LIN {X 0,Y 532.291,Z 792.488,A -85,B 0,C 180,E1 -4217.451,E2 -4217.451} C_VEL
LIN {X 0,Y 532.141,Z 804.373,A -85,B 0,C 180,E1 -4218.078,E2 -4218.078} C_VEL
LIN {X 0,Y 531.859,Z 815.786,A -85,B 0,C 180,E1 -4218.853,E2 -4218.853} C_VEL
LIN {X 0,Y 531.632,Z 825.925,A -85,B 0,C 180,E1 -4219.715,E2 -4219.715} C_VEL
LIN {X 0,Y 531.41,Z 835.007,A -85,B 0,C 180,E1 -4220.672,E2 -4220.672} C_VEL
LIN {X 0,Y 531.158,Z 843.796,A -85,B 0,C 180,E1 -4221.818,E2 -4221.818} C_VEL
LIN {X 0,Y 530.974,Z 851.482,A -85,B 0,C 180,E1 -4223.077,E2 -4223.077} C_VEL
LIN {X 0,Y 530.875,Z 857.285,A -85,B 0,C 180,E1 -4224.297,E2 -4224.297} C_VEL
LIN {X 0,Y 530.745,Z 861.535,A -85,B 0,C 180,E1 -4225.438,E2 -4225.438} C_VEL
LIN {X 0,Y 530.706,Z 863.774,A -85,B 0,C 180,E1 -4226.199,E2 -4226.199} C_VEL
LIN {X 0,Y 530.655,Z 865.602,A -85,B 0,C 180,E1 -4226.958,E2 -4226.958} C_VEL
LIN {X 0,Y 530.61,Z 866.987,A -85,B 0,C 180,E1 -4227.718,E2 -4227.718} C_VEL
LIN {X 0,Y 530.592,Z 868.572,A -85,B 0,C 180,E1 -4229.236,E2 -4229.236} C_VEL
LIN {X 0,Y 530.583,Z 868.809,A -85,B 0,C 180,E1 -4229.995,E2 -4229.995} C_VEL
LIN {X 0,Y 530.623,Z 868.067,A -85,B 0,C 180,E1 -4231.513,E2 -4231.513} C_VEL
LIN {X 0,Y 530.65,Z 865.813,A -85,B 0,C 180,E1 -4233.032,E2 -4233.032} C_VEL
LIN {X 0,Y 530.738,Z 863.013,A -85,B 0,C 180,E1 -4234.171,E2 -4234.171} C_VEL
LIN {X 0,Y 530.785,Z 859.223,A -85,B 0,C 180,E1 -4235.313,E2 -4235.313} C_VEL
LIN {X 0,Y 530.93,Z 853.861,A -85,B 0,C 180,E1 -4236.551,E2 -4236.551} C_VEL
LIN {X 0,Y 531.084,Z 846.949,A -85,B 0,C 180,E1 -4237.79,E2 -4237.79} C_VEL
LIN {X 0,Y 531.313,Z 838.946,A -85,B 0,C 180,E1 -4238.936,E2 -4238.936} C_VEL
LIN {X 0,Y 531.519,Z 830.744,A -85,B 0,C 180,E1 -4239.892,E2 -4239.892} C_VEL
LIN {X 0,Y 531.753,Z 820.601,A -85,B 0,C 180,E1 -4240.85,E2 -4240.85} C_VEL
LIN {X 0,Y 532.059,Z 810.192,A -85,B 0,C 180,E1 -4241.638,E2 -4241.638} C_VEL
LIN {X 0,Y 532.239,Z 798.418,A -85,B 0,C 180,E1 -4242.348,E2 -4242.348} C_VEL
LIN {X 0,Y 532.349,Z 785.959,A -85,B 0,C 180,E1 -4242.91,E2 -4242.91} C_VEL
LIN {X 0,Y 532.464,Z 772.907,A -85,B 0,C 180,E1 -4243.325,E2 -4243.325} C_VEL
LIN {X 0,Y 532.541,Z 760.671,A -85,B 0,C 180,E1 -4243.566,E2 -4243.566} C_VEL
LIN {X 0,Y 532.699,Z 691.55,A -85,B 0,C 180,E1 -4244.506,E2 -4244.506} C_VEL
LIN {X 0,Y 531.049,Z 686.337,A -85,B 0,C 180,E1 -4244.639,E2 -4244.639} C_VEL
LIN {X 0,Y 530.967,Z 686.343,A -85,B 0,C 180,E1 -4247.718,E2 -4247.718} C_VEL
LIN {X 0,Y 531.008,Z 686.337,A -85,B 0,C 180,E1 -4250.121,E2 -4250.121} C_VEL
LIN {X 0,Y 530.923,Z 686.348,A -85,B 0,C 180,E1 -4252.567,E2 -4252.567} C_VEL
LIN {X 0,Y 530.945,Z 686.35,A -85,B 0,C 180,E1 -4255.053,E2 -4255.053} C_VEL
LIN {X 0,Y 530.984,Z 686.34,A -85,B 0,C 180,E1 -4257.589,E2 -4257.589} C_VEL
LIN {X 0,Y 530.943,Z 686.344,A -85,B 0,C 180,E1 -4260.639,E2 -4260.639} C_VEL
LIN {X 0,Y 530.955,Z 686.344,A -85,B 0,C 180,E1 -4263.766,E2 -4263.766} C_VEL
LIN {X 0,Y 530.927,Z 686.345,A -85,B 0,C 180,E1 -4266.552,E2 -4266.552} C_VEL
LIN {X 0,Y 530.964,Z 686.345,A -85,B 0,C 180,E1 -4269.851,E2 -4269.851} C_VEL
LIN {X 0,Y 530.941,Z 686.344,A -85,B 0,C 180,E1 -4272.45,E2 -4272.45} C_VEL
LIN {X 0,Y 530.937,Z 686.346,A -85,B 0,C 180,E1 -4275.615,E2 -4275.615} C_VEL
LIN {X 0,Y 530.968,Z 686.341,A -85,B 0,C 180,E1 -4278.562,E2 -4278.562} C_VEL
LIN {X 0,Y 530.97,Z 686.339,A -85,B 0,C 180,E1 -4280.555,E2 -4280.555} C_VEL
LIN {X 0,Y 530.915,Z 686.355,A -85,B 0,C 180,E1 -4283.837,E2 -4283.837} C_VEL
LIN {X 0,Y 530.938,Z 686.345,A -85,B 0,C 180,E1 -4286.489,E2 -4286.489} C_VEL
LIN {X 0,Y 530.946,Z 686.342,A -85,B 0,C 180,E1 -4289.344,E2 -4289.344} C_VEL
LIN {X 0,Y 530.953,Z 686.347,A -85,B 0,C 180,E1 -4292.462,E2 -4292.462} C_VEL
LIN {X 0,Y 530.958,Z 686.341,A -85,B 0,C 180,E1 -4294.94,E2 -4294.94} C_VEL
LIN {X 0,Y 530.91,Z 686.353,A -85,B 0,C 180,E1 -4298.244,E2 -4298.244} C_VEL
LIN {X 0,Y 530.925,Z 686.349,A -85,B 0,C 180,E1 -4300.675,E2 -4300.675} C_VEL
LIN {X 0,Y 530.926,Z 686.344,A -85,B 0,C 180,E1 -4303.069,E2 -4303.069} C_VEL
LIN {X 0,Y 530.975,Z 686.339,A -85,B 0,C 180,E1 -4305.435,E2 -4305.435} C_VEL
LIN {X 0,Y 530.983,Z 686.345,A -85,B 0,C 180,E1 -4308.548,E2 -4308.548} C_VEL
LIN {X 0,Y 530.989,Z 686.337,A -85,B 0,C 180,E1 -4311.628,E2 -4311.628} C_VEL
LIN {X 0,Y 531.075,Z 686.334,A -85,B 0,C 180,E1 -4314.685,E2 -4314.685} C_VEL
LIN {X 0,Y 531.061,Z 686.328,A -85,B 0,C 180,E1 -4317.725,E2 -4317.725} C_VEL
LIN {X 0,Y 531.084,Z 686.332,A -85,B 0,C 180,E1 -4320.758,E2 -4320.758} C_VEL
LIN {X 0,Y 531.043,Z 686.337,A -85,B 0,C 180,E1 -4323.034,E2 -4323.034} C_VEL
LIN {X 0,Y 531.015,Z 686.335,A -85,B 0,C 180,E1 -4326.078,E2 -4326.078} C_VEL
LIN {X 0,Y 530.969,Z 686.346,A -85,B 0,C 180,E1 -4329.139,E2 -4329.139} C_VEL
LIN {X 0,Y 530.989,Z 686.342,A -85,B 0,C 180,E1 -4331.683,E2 -4331.683} C_VEL
LIN {X 0,Y 530.972,Z 686.342,A -85,B 0,C 180,E1 -4334.966,E2 -4334.966} C_VEL
LIN {X 0,Y 530.944,Z 686.349,A -85,B 0,C 180,E1 -4337.725,E2 -4337.725} C_VEL
LIN {X 0,Y 530.933,Z 686.342,A -85,B 0,C 180,E1 -4340.941,E2 -4340.941} C_VEL
LIN {X 0,Y 530.958,Z 686.342,A -85,B 0,C 180,E1 -4344.226,E2 -4344.226} C_VEL
LIN {X 0,Y 530.956,Z 686.34,A -85,B 0,C 180,E1 -4346.746,E2 -4346.746} C_VEL
LIN {X 0,Y 530.935,Z 686.345,A -85,B 0,C 180,E1 -4349.326,E2 -4349.326} C_VEL
LIN {X 0,Y 530.92,Z 686.353,A -85,B 0,C 180,E1 -4352.108,E2 -4352.108} C_VEL
LIN {X 0,Y 530.93,Z 686.344,A -85,B 0,C 180,E1 -4354.859,E2 -4354.859} C_VEL
LIN {X 0,Y 530.911,Z 686.348,A -85,B 0,C 180,E1 -4357.512,E2 -4357.512} C_VEL
LIN {X 0,Y 530.981,Z 686.344,A -85,B 0,C 180,E1 -4360.433,E2 -4360.433} C_VEL
LIN {X 0,Y 530.917,Z 686.347,A -85,B 0,C 180,E1 -4363.5,E2 -4363.5} C_VEL
LIN {X 0,Y 530.918,Z 686.352,A -85,B 0,C 180,E1 -4366.511,E2 -4366.511} C_VEL
LIN {X 0,Y 530.966,Z 686.341,A -85,B 0,C 180,E1 -4369.576,E2 -4369.576} C_VEL
LIN {X 0,Y 530.928,Z 686.353,A -85,B 0,C 180,E1 -4372.583,E2 -4372.583} C_VEL
LIN {X 0,Y 530.962,Z 686.34,A -85,B 0,C 180,E1 -4375.317,E2 -4375.317} C_VEL
LIN {X 0,Y 530.934,Z 686.348,A -85,B 0,C 180,E1 -4378.038,E2 -4378.038} C_VEL
LIN {X 0,Y 530.962,Z 686.35,A -85,B 0,C 180,E1 -4381.139,E2 -4381.139} C_VEL
LIN {X 0,Y 531.008,Z 686.532,A -85,B 0,C 180,E1 -4381.45,E2 -4381.45} C_VEL
LIN {X 0,Y 533.727,Z 698.362,A -85,B 0,C 180,E1 -4382.988,E2 -4382.988} C_VEL
LIN {X 0,Y 533.507,Z 718.499,A -85,B 0,C 180,E1 -4385.361,E2 -4385.361} C_VEL
LIN {X 0,Y 532.997,Z 742.504,A -85,B 0,C 180,E1 -4388.137,E2 -4388.137} C_VEL
LIN {X 0,Y 532.397,Z 768.598,A -85,B 0,C 180,E1 -4391.137,E2 -4391.137} C_VEL
LIN {X 0,Y 531.853,Z 792.13,A -85,B 0,C 180,E1 -4393.895,E2 -4393.895} C_VEL
LIN {X 0,Y 531.68,Z 801.876,A -85,B 0,C 180,E1 -4395.029,E2 -4395.029} C_VEL
LIN {X 0,Y 532.81,Z 811.855,A -85,B 0,C 180,E1 -4395.201,E2 -4395.201} C_VEL
LIN {X 0,Y 532.375,Z 912.231,A -85,B 0,C 180,E1 -4396.576,E2 -4396.576} C_VEL
LIN {X 0,Y 532.216,Z 925.399,A -85,B 0,C 180,E1 -4396.912,E2 -4396.912} C_VEL
LIN {X 0,Y 531.975,Z 937.504,A -85,B 0,C 180,E1 -4397.367,E2 -4397.367} C_VEL
LIN {X 0,Y 531.811,Z 948.839,A -85,B 0,C 180,E1 -4397.94,E2 -4397.94} C_VEL
LIN {X 0,Y 531.567,Z 959.985,A -85,B 0,C 180,E1 -4398.664,E2 -4398.664} C_VEL
LIN {X 0,Y 531.26,Z 970.602,A -85,B 0,C 180,E1 -4399.526,E2 -4399.526} C_VEL
LIN {X 0,Y 531.062,Z 980.153,A -85,B 0,C 180,E1 -4400.484,E2 -4400.484} C_VEL
LIN {X 0,Y 530.885,Z 988.003,A -85,B 0,C 180,E1 -4401.441,E2 -4401.441} C_VEL
LIN {X 0,Y 530.684,Z 995.655,A -85,B 0,C 180,E1 -4402.587,E2 -4402.587} C_VEL
LIN {X 0,Y 530.599,Z 1002.705,A -85,B 0,C 180,E1 -4403.923,E2 -4403.923} C_VEL
LIN {X 0,Y 530.457,Z 1007.392,A -85,B 0,C 180,E1 -4405.065,E2 -4405.065} C_VEL
LIN {X 0,Y 530.514,Z 1010.975,A -85,B 0,C 180,E1 -4406.207,E2 -4406.207} C_VEL
LIN {X 0,Y 530.456,Z 1012.821,A -85,B 0,C 180,E1 -4406.967,E2 -4406.967} C_VEL
LIN {X 0,Y 530.409,Z 1014.205,A -85,B 0,C 180,E1 -4407.727,E2 -4407.727} C_VEL
LIN {X 0,Y 530.344,Z 1015.789,A -85,B 0,C 180,E1 -4409.246,E2 -4409.246} C_VEL
LIN {X 0,Y 530.342,Z 1016,A -85,B 0,C 180,E1 -4410.005,E2 -4410.005} C_VEL
LIN {X 0,Y 530.361,Z 1015.178,A -85,B 0,C 180,E1 -4411.524,E2 -4411.524} C_VEL
LIN {X 0,Y 530.411,Z 1014.188,A -85,B 0,C 180,E1 -4412.283,E2 -4412.283} C_VEL
LIN {X 0,Y 530.458,Z 1012.797,A -85,B 0,C 180,E1 -4413.043,E2 -4413.043} C_VEL
LIN {X 0,Y 530.524,Z 1009.881,A -85,B 0,C 180,E1 -4414.183,E2 -4414.183} C_VEL
LIN {X 0,Y 530.526,Z 1005.932,A -85,B 0,C 180,E1 -4415.325,E2 -4415.325} C_VEL
LIN {X 0,Y 530.604,Z 1000.238,A -85,B 0,C 180,E1 -4416.587,E2 -4416.587} C_VEL
LIN {X 0,Y 530.763,Z 993.207,A -85,B 0,C 180,E1 -4417.805,E2 -4417.805} C_VEL
LIN {X 0,Y 530.932,Z 984.957,A -85,B 0,C 180,E1 -4418.952,E2 -4418.952} C_VEL
LIN {X 0,Y 531.112,Z 976.496,A -85,B 0,C 180,E1 -4419.91,E2 -4419.91} C_VEL
LIN {X 0,Y 531.415,Z 966.041,A -85,B 0,C 180,E1 -4420.867,E2 -4420.867} C_VEL
LIN {X 0,Y 531.648,Z 955.001,A -85,B 0,C 180,E1 -4421.681,E2 -4421.681} C_VEL
LIN {X 0,Y 531.912,Z 944.33,A -85,B 0,C 180,E1 -4422.306,E2 -4422.306} C_VEL
LIN {X 0,Y 532.097,Z 932.66,A -85,B 0,C 180,E1 -4422.834,E2 -4422.834} C_VEL
LIN {X 0,Y 532.285,Z 919.192,A -85,B 0,C 180,E1 -4423.267,E2 -4423.267} C_VEL
LIN {X 0,Y 532.452,Z 905.789,A -85,B 0,C 180,E1 -4423.53,E2 -4423.53} C_VEL
LIN {X 0,Y 532.775,Z 810.11,A -85,B 0,C 180,E1 -4424.824,E2 -4424.824} C_VEL
LIN {X 0,Y 531.69,Z 801.879,A -85,B 0,C 180,E1 -4424.97,E2 -4424.97} C_VEL
LIN {X 0,Y 532.296,Z 774.205,A -85,B 0,C 180,E1 -4428.201,E2 -4428.201} C_VEL
LIN {X 0,Y 532.732,Z 753.381,A -85,B 0,C 180,E1 -4430.62,E2 -4430.62} C_VEL
LIN {X 0,Y 533.236,Z 730.084,A -85,B 0,C 180,E1 -4433.294,E2 -4433.294} C_VEL
LIN {X 0,Y 533.69,Z 705.785,A -85,B 0,C 180,E1 -4436.131,E2 -4436.131} C_VEL
LIN {X 0,Y 533.739,Z 698.273,A -85,B 0,C 180,E1 -4437.022,E2 -4437.022} C_VEL
LIN {X 0,Y 530.97,Z 686.348,A -85,B 0,C 180,E1 -4438.587,E2 -4438.587} C_VEL
LIN {X 0,Y 530.938,Z 686.353,A -85,B 0,C 180,E1 -4441.084,E2 -4441.084} C_VEL
LIN {X 0,Y 530.897,Z 686.353,A -85,B 0,C 180,E1 -4443.783,E2 -4443.783} C_VEL
LIN {X 0,Y 530.902,Z 686.347,A -85,B 0,C 180,E1 -4446.566,E2 -4446.566} C_VEL
LIN {X 0,Y 530.941,Z 686.349,A -85,B 0,C 180,E1 -4449.451,E2 -4449.451} C_VEL
LIN {X 0,Y 530.917,Z 686.347,A -85,B 0,C 180,E1 -4452.466,E2 -4452.466} C_VEL
LIN {X 0,Y 530.974,Z 686.345,A -85,B 0,C 180,E1 -4455.451,E2 -4455.451} C_VEL
LIN {X 0,Y 530.965,Z 686.342,A -85,B 0,C 180,E1 -4458.561,E2 -4458.561} C_VEL
LIN {X 0,Y 530.96,Z 686.347,A -85,B 0,C 180,E1 -4461.529,E2 -4461.529} C_VEL
LIN {X 0,Y 530.948,Z 686.343,A -85,B 0,C 180,E1 -4464.379,E2 -4464.379} C_VEL
LIN {X 0,Y 530.979,Z 686.346,A -85,B 0,C 180,E1 -4467.134,E2 -4467.134} C_VEL
LIN {X 0,Y 530.965,Z 686.344,A -85,B 0,C 180,E1 -4469.803,E2 -4469.803} C_VEL
LIN {X 0,Y 530.977,Z 686.341,A -85,B 0,C 180,E1 -4472.478,E2 -4472.478} C_VEL
LIN {X 0,Y 530.989,Z 686.342,A -85,B 0,C 180,E1 -4474.942,E2 -4474.942} C_VEL
LIN {X 0,Y 530.982,Z 686.34,A -85,B 0,C 180,E1 -4478.247,E2 -4478.247} C_VEL
LIN {X 0,Y 531.001,Z 686.339,A -85,B 0,C 180,E1 -4480.677,E2 -4480.677} C_VEL
LIN {X 0,Y 530.974,Z 686.346,A -85,B 0,C 180,E1 -4483.071,E2 -4483.071} C_VEL
LIN {X 0,Y 531.031,Z 686.341,A -85,B 0,C 180,E1 -4485.534,E2 -4485.534} C_VEL
LIN {X 0,Y 532.595,Z 691.472,A -85,B 0,C 180,E1 -4485.655,E2 -4485.655} C_VEL
LIN {X 0,Y 532.362,Z 763.672,A -85,B 0,C 180,E1 -4486.667,E2 -4486.667} C_VEL
LIN {X 0,Y 532.273,Z 775.605,A -85,B 0,C 180,E1 -4486.956,E2 -4486.956} C_VEL
LIN {X 0,Y 532.095,Z 785.975,A -85,B 0,C 180,E1 -4487.315,E2 -4487.315} C_VEL
LIN {X 0,Y 531.937,Z 796.416,A -85,B 0,C 180,E1 -4487.796,E2 -4487.796} C_VEL
LIN {X 0,Y 531.787,Z 805.876,A -85,B 0,C 180,E1 -4488.344,E2 -4488.344} C_VEL
LIN {X 0,Y 531.527,Z 815.647,A -85,B 0,C 180,E1 -4489.043,E2 -4489.043} C_VEL
LIN {X 0,Y 531.372,Z 823.465,A -85,B 0,C 180,E1 -4489.715,E2 -4489.715} C_VEL
LIN {X 0,Y 531.113,Z 832.637,A -85,B 0,C 180,E1 -4490.671,E2 -4490.671} C_VEL
LIN {X 0,Y 530.923,Z 840.17,A -85,B 0,C 180,E1 -4491.627,E2 -4491.627} C_VEL
LIN {X 0,Y 530.792,Z 846.415,A -85,B 0,C 180,E1 -4492.583,E2 -4492.583} C_VEL
LIN {X 0,Y 530.69,Z 852.318,A -85,B 0,C 180,E1 -4493.686,E2 -4493.686} C_VEL
LIN {X 0,Y 530.581,Z 856.628,A -85,B 0,C 180,E1 -4494.68,E2 -4494.68} C_VEL
LIN {X 0,Y 530.562,Z 860.504,A -85,B 0,C 180,E1 -4495.822,E2 -4495.822} C_VEL
LIN {X 0,Y 530.499,Z 863.37,A -85,B 0,C 180,E1 -4496.962,E2 -4496.962} C_VEL
LIN {X 0,Y 530.43,Z 864.833,A -85,B 0,C 180,E1 -4497.722,E2 -4497.722} C_VEL
LIN {X 0,Y 530.375,Z 866.384,A -85,B 0,C 180,E1 -4499.241,E2 -4499.241} C_VEL
LIN {X 0,Y 530.371,Z 866.629,A -85,B 0,C 180,E1 -4500,E2 -4500} C_VEL
LIN {X 0,Y 530.384,Z 865.83,A -85,B 0,C 180,E1 -4501.519,E2 -4501.519} C_VEL
LIN {X 0,Y 530.425,Z 864.921,A -85,B 0,C 180,E1 -4502.278,E2 -4502.278} C_VEL
LIN {X 0,Y 530.55,Z 861.742,A -85,B 0,C 180,E1 -4503.798,E2 -4503.798} C_VEL
LIN {X 0,Y 530.524,Z 858.271,A -85,B 0,C 180,E1 -4504.94,E2 -4504.94} C_VEL
LIN {X 0,Y 530.669,Z 853.695,A -85,B 0,C 180,E1 -4506.082,E2 -4506.082} C_VEL
LIN {X 0,Y 530.754,Z 847.914,A -85,B 0,C 180,E1 -4507.227,E2 -4507.227} C_VEL
LIN {X 0,Y 530.91,Z 841.981,A -85,B 0,C 180,E1 -4508.181,E2 -4508.181} C_VEL
LIN {X 0,Y 531.06,Z 834.829,A -85,B 0,C 180,E1 -4509.138,E2 -4509.138} C_VEL
LIN {X 0,Y 531.292,Z 826.099,A -85,B 0,C 180,E1 -4510.095,E2 -4510.095} C_VEL
LIN {X 0,Y 531.474,Z 816.505,A -85,B 0,C 180,E1 -4510.958,E2 -4510.958} C_VEL
LIN {X 0,Y 531.733,Z 807.033,A -85,B 0,C 180,E1 -4511.653,E2 -4511.653} C_VEL
LIN {X 0,Y 531.927,Z 797.845,A -85,B 0,C 180,E1 -4512.204,E2 -4512.204} C_VEL
LIN {X 0,Y 532.049,Z 787.908,A -85,B 0,C 180,E1 -4512.686,E2 -4512.686} C_VEL
LIN {X 0,Y 532.22,Z 777.605,A -85,B 0,C 180,E1 -4513.07,E2 -4513.07} C_VEL
LIN {X 0,Y 532.354,Z 767.993,A -85,B 0,C 180,E1 -4513.334,E2 -4513.334} C_VEL
LIN {X 0,Y 532.42,Z 756.137,A -85,B 0,C 180,E1 -4513.551,E2 -4513.551} C_VEL
LIN {X 0,Y 532.573,Z 691.328,A -85,B 0,C 180,E1 -4514.441,E2 -4514.441} C_VEL
LIN {X 0,Y 531.088,Z 686.334,A -85,B 0,C 180,E1 -4514.562,E2 -4514.562} C_VEL
LIN {X 0,Y 530.993,Z 686.338,A -85,B 0,C 180,E1 -4517.723,E2 -4517.723} C_VEL
LIN {X 0,Y 531.026,Z 686.334,A -85,B 0,C 180,E1 -4520.127,E2 -4520.127} C_VEL
LIN {X 0,Y 530.954,Z 686.348,A -85,B 0,C 180,E1 -4522.573,E2 -4522.573} C_VEL
LIN {X 0,Y 530.99,Z 686.343,A -85,B 0,C 180,E1 -4525.059,E2 -4525.059} C_VEL
LIN {X 0,Y 530.977,Z 686.338,A -85,B 0,C 180,E1 -4527.598,E2 -4527.598} C_VEL
LIN {X 0,Y 530.973,Z 686.34,A -85,B 0,C 180,E1 -4530.197,E2 -4530.197} C_VEL
LIN {X 0,Y 530.97,Z 686.346,A -85,B 0,C 180,E1 -4532.675,E2 -4532.675} C_VEL
LIN {X 0,Y 530.318,Z 686.433,A -85,B 0,C 180,E1 -4533.308,E2 -4533.308} C_VEL
LIN {X 0,Y 527.443,Z 686.788,A -85,B 0,C 180,E1 -4534.335,E2 -4534.335} C_VEL
LIN {X 0,Y 525.01,Z 687.087,A -85,B 0,C 180,E1 -4535.162,E2 -4535.162} C_VEL
LIN {X 0,Y 523.977,Z 687.21,A -85,B 0,C 180,E1 -4535.801,E2 -4535.801} C_VEL
LIN {X 0,Y 523.901,Z 687.219,A -85,B 0,C 180,E1 -4536.018,E2 -4536.018} C_VEL
LIN {X 0,Y 523.926,Z 687.224,A -85,B 0,C 180,E1 -4539.085,E2 -4539.085} C_VEL
LIN {X 0,Y 523.922,Z 687.216,A -85,B 0,C 180,E1 -4542.122,E2 -4542.122} C_VEL
LIN {X 0,Y 523.948,Z 687.218,A -85,B 0,C 180,E1 -4545.31,E2 -4545.31} C_VEL
LIN {X 0,Y 523.93,Z 687.219,A -85,B 0,C 180,E1 -4548.693,E2 -4548.693} C_VEL
LIN {X 0,Y 523.913,Z 687.226,A -85,B 0,C 180,E1 -4551.082,E2 -4551.082} C_VEL
LIN {X 0,Y 523.871,Z 687.224,A -85,B 0,C 180,E1 -4553.82,E2 -4553.82} C_VEL
LIN {X 0,Y 523.91,Z 687.22,A -85,B 0,C 180,E1 -4556.63,E2 -4556.63} C_VEL
LIN {X 0,Y 523.921,Z 687.224,A -85,B 0,C 180,E1 -4559.35,E2 -4559.35} C_VEL
LIN {X 0,Y 523.888,Z 687.221,A -85,B 0,C 180,E1 -4562.301,E2 -4562.301} C_VEL
LIN {X 0,Y 523.901,Z 687.228,A -85,B 0,C 180,E1 -4565.423,E2 -4565.423} C_VEL
LIN {X 0,Y 523.934,Z 687.219,A -85,B 0,C 180,E1 -4567.935,E2 -4567.935} C_VEL
LIN {X 0,Y 523.914,Z 687.22,A -85,B 0,C 180,E1 -4570.402,E2 -4570.402} C_VEL
LIN {X 0,Y 523.942,Z 687.219,A -85,B 0,C 180,E1 -4572.832,E2 -4572.832} C_VEL
LIN {X 0,Y 523.949,Z 687.222,A -85,B 0,C 180,E1 -4575.255,E2 -4575.255} C_VEL
LIN {X 0,Y 526,Z 694.266,A -85,B 0,C 180,E1 -4575.419,E2 -4575.419} C_VEL
LIN {X 0,Y 525.59,Z 767.37,A -85,B 0,C 180,E1 -4576.438,E2 -4576.438} C_VEL
LIN {X 0,Y 525.584,Z 779.802,A -85,B 0,C 180,E1 -4576.758,E2 -4576.758} C_VEL
LIN {X 0,Y 525.469,Z 792.273,A -85,B 0,C 180,E1 -4577.232,E2 -4577.232} C_VEL
LIN {X 0,Y 525.256,Z 802.381,A -85,B 0,C 180,E1 -4577.742,E2 -4577.742} C_VEL
LIN {X 0,Y 525.055,Z 812.897,A -85,B 0,C 180,E1 -4578.413,E2 -4578.413} C_VEL
LIN {X 0,Y 524.798,Z 823.787,A -85,B 0,C 180,E1 -4579.287,E2 -4579.287} C_VEL
LIN {X 0,Y 524.563,Z 832.588,A -85,B 0,C 180,E1 -4580.16,E2 -4580.16} C_VEL
LIN {X 0,Y 524.301,Z 842.098,A -85,B 0,C 180,E1 -4581.322,E2 -4581.322} C_VEL
LIN {X 0,Y 524.056,Z 849.799,A -85,B 0,C 180,E1 -4582.502,E2 -4582.502} C_VEL
LIN {X 0,Y 523.995,Z 855.494,A -85,B 0,C 180,E1 -4583.59,E2 -4583.59} C_VEL
LIN {X 0,Y 523.771,Z 861.247,A -85,B 0,C 180,E1 -4584.992,E2 -4584.992} C_VEL
LIN {X 0,Y 523.693,Z 864.778,A -85,B 0,C 180,E1 -4586.148,E2 -4586.148} C_VEL
LIN {X 0,Y 523.637,Z 866.606,A -85,B 0,C 180,E1 -4586.918,E2 -4586.918} C_VEL
LIN {X 0,Y 523.602,Z 867.989,A -85,B 0,C 180,E1 -4587.687,E2 -4587.687} C_VEL
LIN {X 0,Y 523.581,Z 869.573,A -85,B 0,C 180,E1 -4589.226,E2 -4589.226} C_VEL
LIN {X 0,Y 523.57,Z 869.81,A -85,B 0,C 180,E1 -4589.995,E2 -4589.995} C_VEL
LIN {X 0,Y 523.62,Z 869.066,A -85,B 0,C 180,E1 -4591.533,E2 -4591.533} C_VEL
LIN {X 0,Y 523.631,Z 866.815,A -85,B 0,C 180,E1 -4593.072,E2 -4593.072} C_VEL
LIN {X 0,Y 523.729,Z 864.014,A -85,B 0,C 180,E1 -4594.227,E2 -4594.227} C_VEL
LIN {X 0,Y 523.805,Z 860.221,A -85,B 0,C 180,E1 -4595.384,E2 -4595.384} C_VEL
LIN {X 0,Y 523.958,Z 854.815,A -85,B 0,C 180,E1 -4596.647,E2 -4596.647} C_VEL
LIN {X 0,Y 524.131,Z 847.946,A -85,B 0,C 180,E1 -4597.894,E2 -4597.894} C_VEL
LIN {X 0,Y 524.38,Z 839.943,A -85,B 0,C 180,E1 -4599.055,E2 -4599.055} C_VEL
LIN {X 0,Y 524.603,Z 831.741,A -85,B 0,C 180,E1 -4600.024,E2 -4600.024} C_VEL
LIN {X 0,Y 524.861,Z 821.595,A -85,B 0,C 180,E1 -4600.994,E2 -4600.994} C_VEL
LIN {X 0,Y 525.183,Z 811.163,A -85,B 0,C 180,E1 -4601.794,E2 -4601.794} C_VEL
LIN {X 0,Y 525.378,Z 799.409,A -85,B 0,C 180,E1 -4602.512,E2 -4602.512} C_VEL
LIN {X 0,Y 525.499,Z 786.945,A -85,B 0,C 180,E1 -4603.081,E2 -4603.081} C_VEL
LIN {X 0,Y 525.611,Z 773.889,A -85,B 0,C 180,E1 -4603.502,E2 -4603.502} C_VEL
LIN {X 0,Y 525.687,Z 761.637,A -85,B 0,C 180,E1 -4603.746,E2 -4603.746} C_VEL
LIN {X 0,Y 525.902,Z 693.125,A -85,B 0,C 180,E1 -4604.69,E2 -4604.69} C_VEL
LIN {X 0,Y 523.994,Z 687.217,A -85,B 0,C 180,E1 -4604.833,E2 -4604.833} C_VEL
LIN {X 0,Y 523.933,Z 687.219,A -85,B 0,C 180,E1 -4607.963,E2 -4607.963} C_VEL
LIN {X 0,Y 523.954,Z 687.217,A -85,B 0,C 180,E1 -4610.404,E2 -4610.404} C_VEL
LIN {X 0,Y 523.888,Z 687.227,A -85,B 0,C 180,E1 -4612.887,E2 -4612.887} C_VEL
LIN {X 0,Y 523.89,Z 687.224,A -85,B 0,C 180,E1 -4615.414,E2 -4615.414} C_VEL
LIN {X 0,Y 523.931,Z 687.215,A -85,B 0,C 180,E1 -4617.993,E2 -4617.993} C_VEL
LIN {X 0,Y 523.914,Z 687.222,A -85,B 0,C 180,E1 -4620.848,E2 -4620.848} C_VEL
LIN {X 0,Y 523.926,Z 687.22,A -85,B 0,C 180,E1 -4623.728,E2 -4623.728} C_VEL
LIN {X 0,Y 523.881,Z 687.223,A -85,B 0,C 180,E1 -4626.398,E2 -4626.398} C_VEL
LIN {X 0,Y 523.889,Z 687.22,A -85,B 0,C 180,E1 -4629.078,E2 -4629.078} C_VEL
LIN {X 0,Y 523.92,Z 687.221,A -85,B 0,C 180,E1 -4632.112,E2 -4632.112} C_VEL
LIN {X 0,Y 523.906,Z 687.219,A -85,B 0,C 180,E1 -4635.303,E2 -4635.303} C_VEL
LIN {X 0,Y 523.93,Z 687.217,A -85,B 0,C 180,E1 -4638.681,E2 -4638.681} C_VEL
LIN {X 0,Y 523.906,Z 687.219,A -85,B 0,C 180,E1 -4641.069,E2 -4641.069} C_VEL
LIN {X 0,Y 523.869,Z 687.232,A -85,B 0,C 180,E1 -4643.823,E2 -4643.823} C_VEL
LIN {X 0,Y 523.882,Z 687.223,A -85,B 0,C 180,E1 -4646.631,E2 -4646.631} C_VEL
LIN {X 0,Y 523.925,Z 687.217,A -85,B 0,C 180,E1 -4649.354,E2 -4649.354} C_VEL
LIN {X 0,Y 523.914,Z 687.226,A -85,B 0,C 180,E1 -4652.276,E2 -4652.276} C_VEL
LIN {X 0,Y 523.901,Z 687.223,A -85,B 0,C 180,E1 -4654.578,E2 -4654.578} C_VEL
LIN {X 0,Y 523.851,Z 687.225,A -85,B 0,C 180,E1 -4657.104,E2 -4657.104} C_VEL
LIN {X 0,Y 523.905,Z 687.222,A -85,B 0,C 180,E1 -4659.863,E2 -4659.863} C_VEL
LIN {X 0,Y 523.902,Z 687.222,A -85,B 0,C 180,E1 -4662.835,E2 -4662.835} C_VEL
LIN {X 0,Y 523.942,Z 687.216,A -85,B 0,C 180,E1 -4665.235,E2 -4665.235} C_VEL
LIN {X 0,Y 523.941,Z 687.22,A -85,B 0,C 180,E1 -4668.392,E2 -4668.392} C_VEL
LIN {X 0,Y 523.936,Z 687.216,A -85,B 0,C 180,E1 -4671.515,E2 -4671.515} C_VEL
LIN {X 0,Y 524.032,Z 687.21,A -85,B 0,C 180,E1 -4674.613,E2 -4674.613} C_VEL
LIN {X 0,Y 524.034,Z 687.204,A -85,B 0,C 180,E1 -4677.694,E2 -4677.694} C_VEL
LIN {X 0,Y 524.053,Z 687.208,A -85,B 0,C 180,E1 -4680.768,E2 -4680.768} C_VEL
LIN {X 0,Y 524.009,Z 687.213,A -85,B 0,C 180,E1 -4683.075,E2 -4683.075} C_VEL
LIN {X 0,Y 523.976,Z 687.212,A -85,B 0,C 180,E1 -4686.16,E2 -4686.16} C_VEL
LIN {X 0,Y 523.937,Z 687.222,A -85,B 0,C 180,E1 -4689.263,E2 -4689.263} C_VEL
LIN {X 0,Y 523.946,Z 687.218,A -85,B 0,C 180,E1 -4691.753,E2 -4691.753} C_VEL
LIN {X 0,Y 523.931,Z 687.22,A -85,B 0,C 180,E1 -4695.061,E2 -4695.061} C_VEL
LIN {X 0,Y 523.892,Z 687.224,A -85,B 0,C 180,E1 -4697.972,E2 -4697.972} C_VEL
LIN {X 0,Y 523.9,Z 687.217,A -85,B 0,C 180,E1 -4700.413,E2 -4700.413} C_VEL
LIN {X 0,Y 523.878,Z 687.223,A -85,B 0,C 180,E1 -4702.895,E2 -4702.895} C_VEL
LIN {X 0,Y 523.916,Z 687.222,A -85,B 0,C 180,E1 -4705.421,E2 -4705.421} C_VEL
LIN {X 0,Y 523.905,Z 687.226,A -85,B 0,C 180,E1 -4708.003,E2 -4708.003} C_VEL
LIN {X 0,Y 523.905,Z 687.218,A -85,B 0,C 180,E1 -4710.864,E2 -4710.864} C_VEL
LIN {X 0,Y 523.901,Z 687.225,A -85,B 0,C 180,E1 -4713.74,E2 -4713.74} C_VEL
LIN {X 0,Y 523.864,Z 687.229,A -85,B 0,C 180,E1 -4716.409,E2 -4716.409} C_VEL
LIN {X 0,Y 523.914,Z 687.214,A -85,B 0,C 180,E1 -4719.086,E2 -4719.086} C_VEL
LIN {X 0,Y 523.93,Z 687.217,A -85,B 0,C 180,E1 -4721.319,E2 -4721.319} C_VEL
LIN {X 0,Y 523.906,Z 687.224,A -85,B 0,C 180,E1 -4724.697,E2 -4724.697} C_VEL
LIN {X 0,Y 523.92,Z 687.218,A -85,B 0,C 180,E1 -4727.888,E2 -4727.888} C_VEL
LIN {X 0,Y 523.889,Z 687.226,A -85,B 0,C 180,E1 -4730.922,E2 -4730.922} C_VEL
LIN {X 0,Y 523.886,Z 687.223,A -85,B 0,C 180,E1 -4733.833,E2 -4733.833} C_VEL
LIN {X 0,Y 523.907,Z 687.222,A -85,B 0,C 180,E1 -4736.642,E2 -4736.642} C_VEL
LIN {X 0,Y 523.925,Z 687.223,A -85,B 0,C 180,E1 -4739.362,E2 -4739.362} C_VEL
LIN {X 0,Y 523.947,Z 687.311,A -85,B 0,C 180,E1 -4741.239,E2 -4741.239} C_VEL
LIN {X 0,Y 526.715,Z 699.217,A -85,B 0,C 180,E1 -4742.814,E2 -4742.814} C_VEL
LIN {X 0,Y 526.836,Z 705.601,A -85,B 0,C 180,E1 -4743.59,E2 -4743.59} C_VEL
LIN {X 0,Y 526.382,Z 725.748,A -85,B 0,C 180,E1 -4745.977,E2 -4745.977} C_VEL
LIN {X 0,Y 525.848,Z 750.344,A -85,B 0,C 180,E1 -4748.854,E2 -4748.854} C_VEL
LIN {X 0,Y 525.256,Z 778.435,A -85,B 0,C 180,E1 -4752.083,E2 -4752.083} C_VEL
LIN {X 0,Y 524.739,Z 801.891,A -85,B 0,C 180,E1 -4754.828,E2 -4754.828} C_VEL
LIN {X 0,Y 525.944,Z 811.94,A -85,B 0,C 180,E1 -4755.004,E2 -4755.004} C_VEL
LIN {X 0,Y 525.494,Z 912.231,A -85,B 0,C 180,E1 -4756.397,E2 -4756.397} C_VEL
LIN {X 0,Y 525.294,Z 925.398,A -85,B 0,C 180,E1 -4756.736,E2 -4756.736} C_VEL
LIN {X 0,Y 525.056,Z 937.502,A -85,B 0,C 180,E1 -4757.198,E2 -4757.198} C_VEL
LIN {X 0,Y 524.85,Z 949.633,A -85,B 0,C 180,E1 -4757.825,E2 -4757.825} C_VEL
LIN {X 0,Y 524.549,Z 961.274,A -85,B 0,C 180,E1 -4758.608,E2 -4758.608} C_VEL
LIN {X 0,Y 524.235,Z 971.669,A -85,B 0,C 180,E1 -4759.481,E2 -4759.481} C_VEL
LIN {X 0,Y 524.054,Z 980.161,A -85,B 0,C 180,E1 -4760.355,E2 -4760.355} C_VEL
LIN {X 0,Y 523.85,Z 988.003,A -85,B 0,C 180,E1 -4761.325,E2 -4761.325} C_VEL
LIN {X 0,Y 523.631,Z 995.655,A -85,B 0,C 180,E1 -4762.486,E2 -4762.486} C_VEL
LIN {X 0,Y 523.511,Z 1002.705,A -85,B 0,C 180,E1 -4763.84,E2 -4763.84} C_VEL
LIN {X 0,Y 523.382,Z 1007.392,A -85,B 0,C 180,E1 -4764.998,E2 -4764.998} C_VEL
LIN {X 0,Y 523.442,Z 1010.975,A -85,B 0,C 180,E1 -4766.156,E2 -4766.156} C_VEL
LIN {X 0,Y 523.366,Z 1012.821,A -85,B 0,C 180,E1 -4766.926,E2 -4766.926} C_VEL
LIN {X 0,Y 523.333,Z 1014.204,A -85,B 0,C 180,E1 -4767.696,E2 -4767.696} C_VEL
LIN {X 0,Y 523.25,Z 1015.789,A -85,B 0,C 180,E1 -4769.236,E2 -4769.236} C_VEL
LIN {X 0,Y 523.246,Z 1016,A -85,B 0,C 180,E1 -4770.005,E2 -4770.005} C_VEL
LIN {X 0,Y 523.274,Z 1015.178,A -85,B 0,C 180,E1 -4771.544,E2 -4771.544} C_VEL
LIN {X 0,Y 523.335,Z 1014.187,A -85,B 0,C 180,E1 -4772.314,E2 -4772.314} C_VEL
LIN {X 0,Y 523.368,Z 1012.797,A -85,B 0,C 180,E1 -4773.084,E2 -4773.084} C_VEL
LIN {X 0,Y 523.443,Z 1009.881,A -85,B 0,C 180,E1 -4774.24,E2 -4774.24} C_VEL
LIN {X 0,Y 523.466,Z 1005.932,A -85,B 0,C 180,E1 -4775.397,E2 -4775.397} C_VEL
LIN {X 0,Y 523.528,Z 1000.703,A -85,B 0,C 180,E1 -4776.586,E2 -4776.586} C_VEL
LIN {X 0,Y 523.67,Z 994.437,A -85,B 0,C 180,E1 -4777.717,E2 -4777.717} C_VEL
LIN {X 0,Y 523.857,Z 986.443,A -85,B 0,C 180,E1 -4778.88,E2 -4778.88} C_VEL
LIN {X 0,Y 524.086,Z 978.292,A -85,B 0,C 180,E1 -4779.849,E2 -4779.849} C_VEL
LIN {X 0,Y 524.357,Z 968.35,A -85,B 0,C 180,E1 -4780.82,E2 -4780.82} C_VEL
LIN {X 0,Y 524.636,Z 958.527,A -85,B 0,C 180,E1 -4781.596,E2 -4781.596} C_VEL
LIN {X 0,Y 524.905,Z 946.094,A -85,B 0,C 180,E1 -4782.374,E2 -4782.374} C_VEL
LIN {X 0,Y 525.152,Z 933.882,A -85,B 0,C 180,E1 -4782.958,E2 -4782.958} C_VEL
LIN {X 0,Y 525.367,Z 921.023,A -85,B 0,C 180,E1 -4783.395,E2 -4783.395} C_VEL
LIN {X 0,Y 525.559,Z 907.34,A -85,B 0,C 180,E1 -4783.686,E2 -4783.686} C_VEL
LIN {X 0,Y 525.953,Z 811.558,A -85,B 0,C 180,E1 -4785.001,E2 -4785.001} C_VEL
LIN {X 0,Y 524.756,Z 801.787,A -85,B 0,C 180,E1 -4785.183,E2 -4785.183} C_VEL
LIN {X 0,Y 525.291,Z 776.993,A -85,B 0,C 180,E1 -4788.081,E2 -4788.081} C_VEL
LIN {X 0,Y 525.857,Z 750.272,A -85,B 0,C 180,E1 -4791.156,E2 -4791.156} C_VEL
LIN {X 0,Y 526.35,Z 727.416,A -85,B 0,C 180,E1 -4793.827,E2 -4793.827} C_VEL
LIN {X 0,Y 526.94,Z 702.685,A -85,B 0,C 180,E1 -4796.759,E2 -4796.759} C_VEL
LIN {X 0,Y 526.731,Z 699.131,A -85,B 0,C 180,E1 -4797.196,E2 -4797.196} C_VEL
LIN {X 0,Y 523.938,Z 687.225,A -85,B 0,C 180,E1 -4798.796,E2 -4798.796} C_VEL
LIN {X 0,Y 523.902,Z 687.224,A -85,B 0,C 180,E1 -4801.549,E2 -4801.549} C_VEL
LIN {X 0,Y 523.873,Z 687.227,A -85,B 0,C 180,E1 -4804.298,E2 -4804.298} C_VEL
LIN {X 0,Y 523.852,Z 687.233,A -85,B 0,C 180,E1 -4807.14,E2 -4807.14} C_VEL
LIN {X 0,Y 523.897,Z 687.221,A -85,B 0,C 180,E1 -4810.124,E2 -4810.124} C_VEL
LIN {X 0,Y 523.885,Z 687.231,A -85,B 0,C 180,E1 -4813.174,E2 -4813.174} C_VEL
LIN {X 0,Y 523.931,Z 687.219,A -85,B 0,C 180,E1 -4815.771,E2 -4815.771} C_VEL
LIN {X 0,Y 523.904,Z 687.225,A -85,B 0,C 180,E1 -4818.904,E2 -4818.904} C_VEL
LIN {X 0,Y 523.914,Z 687.22,A -85,B 0,C 180,E1 -4821.898,E2 -4821.898} C_VEL
LIN {X 0,Y 523.928,Z 687.221,A -85,B 0,C 180,E1 -4824.914,E2 -4824.914} C_VEL
LIN {X 0,Y 523.947,Z 687.219,A -85,B 0,C 180,E1 -4827.681,E2 -4827.681} C_VEL
LIN {X 0,Y 523.964,Z 687.215,A -85,B 0,C 180,E1 -4830.678,E2 -4830.678} C_VEL
LIN {X 0,Y 523.939,Z 687.221,A -85,B 0,C 180,E1 -4833.727,E2 -4833.727} C_VEL
LIN {X 0,Y 523.922,Z 687.219,A -85,B 0,C 180,E1 -4836.27,E2 -4836.27} C_VEL
LIN {X 0,Y 523.956,Z 687.217,A -85,B 0,C 180,E1 -4838.767,E2 -4838.767} C_VEL
LIN {X 0,Y 523.956,Z 687.222,A -85,B 0,C 180,E1 -4841.221,E2 -4841.221} C_VEL
LIN {X 0,Y 523.933,Z 687.225,A -85,B 0,C 180,E1 -4843.639,E2 -4843.639} C_VEL
LIN {X 0,Y 523.99,Z 687.219,A -85,B 0,C 180,E1 -4845.354,E2 -4845.354} C_VEL
LIN {X 0,Y 525.785,Z 693.502,A -85,B 0,C 180,E1 -4845.498,E2 -4845.498} C_VEL
LIN {X 0,Y 525.411,Z 765.728,A -85,B 0,C 180,E1 -4846.536,E2 -4846.536} C_VEL
LIN {X 0,Y 525.354,Z 776.619,A -85,B 0,C 180,E1 -4846.806,E2 -4846.806} C_VEL
LIN {X 0,Y 525.22,Z 787.582,A -85,B 0,C 180,E1 -4847.196,E2 -4847.196} C_VEL
LIN {X 0,Y 525.031,Z 797.045,A -85,B 0,C 180,E1 -4847.633,E2 -4847.633} C_VEL
LIN {X 0,Y 524.889,Z 806.735,A -85,B 0,C 180,E1 -4848.198,E2 -4848.198} C_VEL
LIN {X 0,Y 524.619,Z 816.44,A -85,B 0,C 180,E1 -4848.897,E2 -4848.897} C_VEL
LIN {X 0,Y 524.454,Z 824.311,A -85,B 0,C 180,E1 -4849.577,E2 -4849.577} C_VEL
LIN {X 0,Y 524.247,Z 831.9,A -85,B 0,C 180,E1 -4850.353,E2 -4850.353} C_VEL
LIN {X 0,Y 524.052,Z 839.735,A -85,B 0,C 180,E1 -4851.323,E2 -4851.323} C_VEL
LIN {X 0,Y 523.886,Z 846.242,A -85,B 0,C 180,E1 -4852.29,E2 -4852.29} C_VEL
LIN {X 0,Y 523.762,Z 851.416,A -85,B 0,C 180,E1 -4853.204,E2 -4853.204} C_VEL
LIN {X 0,Y 523.72,Z 856.153,A -85,B 0,C 180,E1 -4854.224,E2 -4854.224} C_VEL
LIN {X 0,Y 523.538,Z 860.427,A -85,B 0,C 180,E1 -4855.38,E2 -4855.38} C_VEL
LIN {X 0,Y 523.543,Z 862.605,A -85,B 0,C 180,E1 -4856.151,E2 -4856.151} C_VEL
LIN {X 0,Y 523.437,Z 865.872,A -85,B 0,C 180,E1 -4857.692,E2 -4857.692} C_VEL
LIN {X 0,Y 523.383,Z 867.435,A -85,B 0,C 180,E1 -4859.231,E2 -4859.231} C_VEL
LIN {X 0,Y 523.35,Z 867.66,A -85,B 0,C 180,E1 -4860,E2 -4860} C_VEL
LIN {X 0,Y 523.381,Z 867.463,A -85,B 0,C 180,E1 -4860.769,E2 -4860.769} C_VEL
LIN {X 0,Y 523.4,Z 865.91,A -85,B 0,C 180,E1 -4862.309,E2 -4862.309} C_VEL
LIN {X 0,Y 523.534,Z 862.731,A -85,B 0,C 180,E1 -4863.849,E2 -4863.849} C_VEL
LIN {X 0,Y 523.527,Z 859.234,A -85,B 0,C 180,E1 -4865.006,E2 -4865.006} C_VEL
LIN {X 0,Y 523.671,Z 854.611,A -85,B 0,C 180,E1 -4866.164,E2 -4866.164} C_VEL
LIN {X 0,Y 523.779,Z 848.744,A -85,B 0,C 180,E1 -4867.323,E2 -4867.323} C_VEL
LIN {X 0,Y 523.925,Z 842.771,A -85,B 0,C 180,E1 -4868.291,E2 -4868.291} C_VEL
LIN {X 0,Y 524.098,Z 835.552,A -85,B 0,C 180,E1 -4869.26,E2 -4869.26} C_VEL
LIN {X 0,Y 524.271,Z 828.728,A -85,B 0,C 180,E1 -4870.036,E2 -4870.036} C_VEL
LIN {X 0,Y 524.501,Z 819.464,A -85,B 0,C 180,E1 -4870.91,E2 -4870.91} C_VEL
LIN {X 0,Y 524.724,Z 810.785,A -85,B 0,C 180,E1 -4871.59,E2 -4871.59} C_VEL
LIN {X 0,Y 524.941,Z 801.049,A -85,B 0,C 180,E1 -4872.216,E2 -4872.216} C_VEL
LIN {X 0,Y 525.124,Z 791.591,A -85,B 0,C 180,E1 -4872.709,E2 -4872.709} C_VEL
LIN {X 0,Y 525.339,Z 780.729,A -85,B 0,C 180,E1 -4873.146,E2 -4873.146} C_VEL
LIN {X 0,Y 525.423,Z 769.969,A -85,B 0,C 180,E1 -4873.463,E2 -4873.463} C_VEL
LIN {X 0,Y 525.499,Z 757.157,A -85,B 0,C 180,E1 -4873.708,E2 -4873.708} C_VEL
LIN {X 0,Y 525.662,Z 692.499,A -85,B 0,C 180,E1 -4874.615,E2 -4874.615} C_VEL
LIN {X 0,Y 524.034,Z 687.213,A -85,B 0,C 180,E1 -4874.763,E2 -4874.763} C_VEL
LIN {X 0,Y 523.959,Z 687.215,A -85,B 0,C 180,E1 -4877.969,E2 -4877.969} C_VEL
LIN {X 0,Y 523.964,Z 687.217,A -85,B 0,C 180,E1 -4880.41,E2 -4880.41} C_VEL
LIN {X 0,Y 523.92,Z 687.226,A -85,B 0,C 180,E1 -4882.893,E2 -4882.893} C_VEL
LIN {X 0,Y 523.932,Z 687.218,A -85,B 0,C 180,E1 -4885.42,E2 -4885.42} C_VEL
LIN {X 0,Y 523.928,Z 687.216,A -85,B 0,C 180,E1 -4888.002,E2 -4888.002} C_VEL
LIN {X 0,Y 523.953,Z 687.222,A -85,B 0,C 180,E1 -4890.853,E2 -4890.853} C_VEL
LIN {X 0,Y 523.94,Z 687.215,A -85,B 0,C 180,E1 -4893.728,E2 -4893.728} C_VEL
LIN {X 0,Y 523.901,Z 687.219,A -85,B 0,C 180,E1 -4896.018,E2 -4896.018} C_VEL
LIN {X 0,Y 523.258,Z 687.306,A -85,B 0,C 180,E1 -4896.659,E2 -4896.659} C_VEL
LIN {X 0,Y 520.426,Z 687.66,A -85,B 0,C 180,E1 -4897.701,E2 -4897.701} C_VEL
LIN {X 0,Y 518.013,Z 687.962,A -85,B 0,C 180,E1 -4898.54,E2 -4898.54} C_VEL
LIN {X 0,Y 516.968,Z 688.089,A -85,B 0,C 180,E1 -4899.188,E2 -4899.188} C_VEL
LIN {X 0,Y 516.878,Z 688.098,A -85,B 0,C 180,E1 -4899.407,E2 -4899.407} C_VEL
LIN {X 0,Y 516.898,Z 688.092,A -85,B 0,C 180,E1 -4901.777,E2 -4901.777} C_VEL
LIN {X 0,Y 516.912,Z 688.098,A -85,B 0,C 180,E1 -4905.005,E2 -4905.005} C_VEL
LIN {X 0,Y 516.866,Z 688.096,A -85,B 0,C 180,E1 -4908.405,E2 -4908.405} C_VEL
LIN {X 0,Y 516.877,Z 688.101,A -85,B 0,C 180,E1 -4911.28,E2 -4911.28} C_VEL
LIN {X 0,Y 516.843,Z 688.101,A -85,B 0,C 180,E1 -4914.675,E2 -4914.675} C_VEL
LIN {X 0,Y 516.878,Z 688.099,A -85,B 0,C 180,E1 -4917.46,E2 -4917.46} C_VEL
LIN {X 0,Y 516.852,Z 688.098,A -85,B 0,C 180,E1 -4920.489,E2 -4920.489} C_VEL
LIN {X 0,Y 516.83,Z 688.109,A -85,B 0,C 180,E1 -4923.333,E2 -4923.333} C_VEL
LIN {X 0,Y 516.879,Z 688.097,A -85,B 0,C 180,E1 -4925.923,E2 -4925.923} C_VEL
LIN {X 0,Y 516.861,Z 688.099,A -85,B 0,C 180,E1 -4928.457,E2 -4928.457} C_VEL
LIN {X 0,Y 516.859,Z 688.103,A -85,B 0,C 180,E1 -4930.949,E2 -4930.949} C_VEL
LIN {X 0,Y 516.88,Z 688.104,A -85,B 0,C 180,E1 -4933.405,E2 -4933.405} C_VEL
LIN {X 0,Y 516.901,Z 688.099,A -85,B 0,C 180,E1 -4935.05,E2 -4935.05} C_VEL
LIN {X 0,Y 519.16,Z 695.32,A -85,B 0,C 180,E1 -4935.223,E2 -4935.223} C_VEL
LIN {X 0,Y 518.727,Z 768.406,A -85,B 0,C 180,E1 -4936.255,E2 -4936.255} C_VEL
LIN {X 0,Y 518.759,Z 781.576,A -85,B 0,C 180,E1 -4936.605,E2 -4936.605} C_VEL
LIN {X 0,Y 518.586,Z 794.52,A -85,B 0,C 180,E1 -4937.114,E2 -4937.114} C_VEL
LIN {X 0,Y 518.395,Z 806.418,A -85,B 0,C 180,E1 -4937.759,E2 -4937.759} C_VEL
LIN {X 0,Y 518.077,Z 817.808,A -85,B 0,C 180,E1 -4938.552,E2 -4938.552} C_VEL
LIN {X 0,Y 517.829,Z 827.94,A -85,B 0,C 180,E1 -4939.438,E2 -4939.438} C_VEL
LIN {X 0,Y 517.565,Z 837.019,A -85,B 0,C 180,E1 -4940.42,E2 -4940.42} C_VEL
LIN {X 0,Y 517.26,Z 845.808,A -85,B 0,C 180,E1 -4941.597,E2 -4941.597} C_VEL
LIN {X 0,Y 517.024,Z 853.493,A -85,B 0,C 180,E1 -4942.889,E2 -4942.889} C_VEL
LIN {X 0,Y 516.919,Z 859.292,A -85,B 0,C 180,E1 -4944.143,E2 -4944.143} C_VEL
LIN {X 0,Y 516.731,Z 863.545,A -85,B 0,C 180,E1 -4945.314,E2 -4945.314} C_VEL
LIN {X 0,Y 516.681,Z 865.783,A -85,B 0,C 180,E1 -4946.095,E2 -4946.095} C_VEL
LIN {X 0,Y 516.618,Z 867.61,A -85,B 0,C 180,E1 -4946.876,E2 -4946.876} C_VEL
LIN {X 0,Y 516.593,Z 868.99,A -85,B 0,C 180,E1 -4947.656,E2 -4947.656} C_VEL
LIN {X 0,Y 516.569,Z 870.574,A -85,B 0,C 180,E1 -4949.215,E2 -4949.215} C_VEL
LIN {X 0,Y 516.555,Z 870.811,A -85,B 0,C 180,E1 -4949.995,E2 -4949.995} C_VEL
LIN {X 0,Y 516.615,Z 870.065,A -85,B 0,C 180,E1 -4951.554,E2 -4951.554} C_VEL
LIN {X 0,Y 516.612,Z 867.816,A -85,B 0,C 180,E1 -4953.114,E2 -4953.114} C_VEL
LIN {X 0,Y 516.721,Z 865.015,A -85,B 0,C 180,E1 -4954.285,E2 -4954.285} C_VEL
LIN {X 0,Y 516.823,Z 861.219,A -85,B 0,C 180,E1 -4955.457,E2 -4955.457} C_VEL
LIN {X 0,Y 516.984,Z 855.786,A -85,B 0,C 180,E1 -4956.743,E2 -4956.743} C_VEL
LIN {X 0,Y 517.175,Z 848.944,A -85,B 0,C 180,E1 -4958.001,E2 -4958.001} C_VEL
LIN {X 0,Y 517.448,Z 840.94,A -85,B 0,C 180,E1 -4959.177,E2 -4959.177} C_VEL
LIN {X 0,Y 517.69,Z 832.737,A -85,B 0,C 180,E1 -4960.159,E2 -4960.159} C_VEL
LIN {X 0,Y 517.968,Z 822.59,A -85,B 0,C 180,E1 -4961.142,E2 -4961.142} C_VEL
LIN {X 0,Y 518.318,Z 812.153,A -85,B 0,C 180,E1 -4961.953,E2 -4961.953} C_VEL
LIN {X 0,Y 518.508,Z 800.92,A -85,B 0,C 180,E1 -4962.651,E2 -4962.651} C_VEL
LIN {X 0,Y 518.644,Z 789.094,A -85,B 0,C 180,E1 -4963.212,E2 -4963.212} C_VEL
LIN {X 0,Y 518.77,Z 775.778,A -85,B 0,C 180,E1 -4963.658,E2 -4963.658} C_VEL
LIN {X 0,Y 518.825,Z 764.109,A -85,B 0,C 180,E1 -4963.906,E2 -4963.906} C_VEL
LIN {X 0,Y 519.107,Z 694.689,A -85,B 0,C 180,E1 -4964.878,E2 -4964.878} C_VEL
LIN {X 0,Y 516.969,Z 688.093,A -85,B 0,C 180,E1 -4965.041,E2 -4965.041} C_VEL
LIN {X 0,Y 516.901,Z 688.097,A -85,B 0,C 180,E1 -4968.216,E2 -4968.216} C_VEL
LIN {X 0,Y 516.894,Z 688.101,A -85,B 0,C 180,E1 -4970.695,E2 -4970.695} C_VEL
LIN {X 0,Y 516.864,Z 688.096,A -85,B 0,C 180,E1 -4974.067,E2 -4974.067} C_VEL
LIN {X 0,Y 516.883,Z 688.095,A -85,B 0,C 180,E1 -4976.652,E2 -4976.652} C_VEL
LIN {X 0,Y 516.881,Z 688.099,A -85,B 0,C 180,E1 -4979.517,E2 -4979.517} C_VEL
LIN {X 0,Y 516.863,Z 688.098,A -85,B 0,C 180,E1 -4982.537,E2 -4982.537} C_VEL
LIN {X 0,Y 516.844,Z 688.108,A -85,B 0,C 180,E1 -4985.326,E2 -4985.326} C_VEL
LIN {X 0,Y 516.84,Z 688.096,A -85,B 0,C 180,E1 -4987.937,E2 -4987.937} C_VEL
LIN {X 0,Y 516.865,Z 688.098,A -85,B 0,C 180,E1 -4990.733,E2 -4990.733} C_VEL
LIN {X 0,Y 516.835,Z 688.101,A -85,B 0,C 180,E1 -4993.897,E2 -4993.897} C_VEL
LIN {X 0,Y 516.832,Z 688.102,A -85,B 0,C 180,E1 -4996.101,E2 -4996.101} C_VEL
LIN {X 0,Y 516.865,Z 688.1,A -85,B 0,C 180,E1 -4999.256,E2 -4999.256} C_VEL
LIN {X 0,Y 516.829,Z 688.108,A -85,B 0,C 180,E1 -5002.051,E2 -5002.051} C_VEL
LIN {X 0,Y 516.836,Z 688.099,A -85,B 0,C 180,E1 -5005.171,E2 -5005.171} C_VEL
LIN {X 0,Y 516.823,Z 688.109,A -85,B 0,C 180,E1 -5007.971,E2 -5007.971} C_VEL
LIN {X 0,Y 516.871,Z 688.094,A -85,B 0,C 180,E1 -5010.692,E2 -5010.692} C_VEL
LIN {X 0,Y 516.883,Z 688.097,A -85,B 0,C 180,E1 -5013.798,E2 -5013.798} C_VEL
LIN {X 0,Y 516.807,Z 688.105,A -85,B 0,C 180,E1 -5016.773,E2 -5016.773} C_VEL
LIN {X 0,Y 516.866,Z 688.097,A -85,B 0,C 180,E1 -5019.728,E2 -5019.728} C_VEL
LIN {X 0,Y 516.86,Z 688.102,A -85,B 0,C 180,E1 -5022.594,E2 -5022.594} C_VEL
LIN {X 0,Y 516.888,Z 688.097,A -85,B 0,C 180,E1 -5025.028,E2 -5025.028} C_VEL
LIN {X 0,Y 516.926,Z 688.092,A -85,B 0,C 180,E1 -5028.233,E2 -5028.233} C_VEL
LIN {X 0,Y 516.9,Z 688.094,A -85,B 0,C 180,E1 -5031.398,E2 -5031.398} C_VEL
LIN {X 0,Y 516.992,Z 688.086,A -85,B 0,C 180,E1 -5034.54,E2 -5034.54} C_VEL
LIN {X 0,Y 517.007,Z 688.08,A -85,B 0,C 180,E1 -5037.663,E2 -5037.663} C_VEL
LIN {X 0,Y 517.023,Z 688.084,A -85,B 0,C 180,E1 -5040.779,E2 -5040.779} C_VEL
LIN {X 0,Y 516.976,Z 688.089,A -85,B 0,C 180,E1 -5043.117,E2 -5043.117} C_VEL
LIN {X 0,Y 516.938,Z 688.088,A -85,B 0,C 180,E1 -5046.244,E2 -5046.244} C_VEL
LIN {X 0,Y 516.892,Z 688.099,A -85,B 0,C 180,E1 -5049.39,E2 -5049.39} C_VEL
LIN {X 0,Y 516.905,Z 688.095,A -85,B 0,C 180,E1 -5051.826,E2 -5051.826} C_VEL
LIN {X 0,Y 516.882,Z 688.099,A -85,B 0,C 180,E1 -5055.155,E2 -5055.155} C_VEL
LIN {X 0,Y 516.854,Z 688.099,A -85,B 0,C 180,E1 -5058.225,E2 -5058.225} C_VEL
LIN {X 0,Y 516.842,Z 688.096,A -85,B 0,C 180,E1 -5060.704,E2 -5060.704} C_VEL
LIN {X 0,Y 516.829,Z 688.103,A -85,B 0,C 180,E1 -5063.226,E2 -5063.226} C_VEL
LIN {X 0,Y 516.882,Z 688.096,A -85,B 0,C 180,E1 -5066.202,E2 -5066.202} C_VEL
LIN {X 0,Y 516.87,Z 688.097,A -85,B 0,C 180,E1 -5069.308,E2 -5069.308} C_VEL
LIN {X 0,Y 516.839,Z 688.101,A -85,B 0,C 180,E1 -5072.549,E2 -5072.549} C_VEL
LIN {X 0,Y 516.823,Z 688.102,A -85,B 0,C 180,E1 -5075.337,E2 -5075.337} C_VEL
LIN {X 0,Y 516.828,Z 688.107,A -85,B 0,C 180,E1 -5077.949,E2 -5077.949} C_VEL
LIN {X 0,Y 516.864,Z 688.099,A -85,B 0,C 180,E1 -5080.744,E2 -5080.744} C_VEL
LIN {X 0,Y 516.832,Z 688.105,A -85,B 0,C 180,E1 -5083.909,E2 -5083.909} C_VEL
LIN {X 0,Y 516.835,Z 688.106,A -85,B 0,C 180,E1 -5086.113,E2 -5086.113} C_VEL
LIN {X 0,Y 516.865,Z 688.098,A -85,B 0,C 180,E1 -5089.267,E2 -5089.267} C_VEL
LIN {X 0,Y 516.823,Z 688.108,A -85,B 0,C 180,E1 -5092.28,E2 -5092.28} C_VEL
LIN {X 0,Y 516.857,Z 688.098,A -85,B 0,C 180,E1 -5095.182,E2 -5095.182} C_VEL
LIN {X 0,Y 516.841,Z 688.104,A -85,B 0,C 180,E1 -5097.981,E2 -5097.981} C_VEL
LIN {X 0,Y 516.887,Z 688.171,A -85,B 0,C 180,E1 -5101.036,E2 -5101.036} C_VEL
LIN {X 0,Y 519.912,Z 701.398,A -85,B 0,C 180,E1 -5102.809,E2 -5102.809} C_VEL
LIN {X 0,Y 519.647,Z 720.14,A -85,B 0,C 180,E1 -5105.079,E2 -5105.079} C_VEL
LIN {X 0,Y 519.043,Z 744.176,A -85,B 0,C 180,E1 -5107.937,E2 -5107.937} C_VEL
LIN {X 0,Y 518.384,Z 770.472,A -85,B 0,C 180,E1 -5111.018,E2 -5111.018} C_VEL
LIN {X 0,Y 517.881,Z 793.196,A -85,B 0,C 180,E1 -5113.651,E2 -5113.651} C_VEL
LIN {X 0,Y 517.768,Z 801.616,A -85,B 0,C 180,E1 -5114.623,E2 -5114.623} C_VEL
LIN {X 0,Y 519.085,Z 812.585,A -85,B 0,C 180,E1 -5114.814,E2 -5114.814} C_VEL
LIN {X 0,Y 518.618,Z 912.23,A -85,B 0,C 180,E1 -5116.213,E2 -5116.213} C_VEL
LIN {X 0,Y 518.382,Z 925.397,A -85,B 0,C 180,E1 -5116.556,E2 -5116.556} C_VEL
LIN {X 0,Y 518.134,Z 937.501,A -85,B 0,C 180,E1 -5117.024,E2 -5117.024} C_VEL
LIN {X 0,Y 517.896,Z 949.724,A -85,B 0,C 180,E1 -5117.665,E2 -5117.665} C_VEL
LIN {X 0,Y 517.581,Z 961.273,A -85,B 0,C 180,E1 -5118.453,E2 -5118.453} C_VEL
LIN {X 0,Y 517.224,Z 971.669,A -85,B 0,C 180,E1 -5119.337,E2 -5119.337} C_VEL
LIN {X 0,Y 517.049,Z 980.166,A -85,B 0,C 180,E1 -5120.224,E2 -5120.224} C_VEL
LIN {X 0,Y 516.812,Z 988.003,A -85,B 0,C 180,E1 -5121.206,E2 -5121.206} C_VEL
LIN {X 0,Y 516.577,Z 995.655,A -85,B 0,C 180,E1 -5122.383,E2 -5122.383} C_VEL
LIN {X 0,Y 516.416,Z 1002.704,A -85,B 0,C 180,E1 -5123.755,E2 -5123.755} C_VEL
LIN {X 0,Y 516.311,Z 1007.392,A -85,B 0,C 180,E1 -5124.93,E2 -5124.93} C_VEL
LIN {X 0,Y 516.353,Z 1010.975,A -85,B 0,C 180,E1 -5126.103,E2 -5126.103} C_VEL
LIN {X 0,Y 516.281,Z 1012.821,A -85,B 0,C 180,E1 -5126.884,E2 -5126.884} C_VEL
LIN {X 0,Y 516.26,Z 1014.204,A -85,B 0,C 180,E1 -5127.665,E2 -5127.665} C_VEL
LIN {X 0,Y 516.16,Z 1015.789,A -85,B 0,C 180,E1 -5129.225,E2 -5129.225} C_VEL
LIN {X 0,Y 516.154,Z 1016,A -85,B 0,C 180,E1 -5130.005,E2 -5130.005} C_VEL
LIN {X 0,Y 516.192,Z 1015.177,A -85,B 0,C 180,E1 -5131.565,E2 -5131.565} C_VEL
LIN {X 0,Y 516.261,Z 1014.186,A -85,B 0,C 180,E1 -5132.346,E2 -5132.346} C_VEL
LIN {X 0,Y 516.284,Z 1012.797,A -85,B 0,C 180,E1 -5133.126,E2 -5133.126} C_VEL
LIN {X 0,Y 516.345,Z 1009.881,A -85,B 0,C 180,E1 -5134.298,E2 -5134.298} C_VEL
LIN {X 0,Y 516.407,Z 1005.932,A -85,B 0,C 180,E1 -5135.471,E2 -5135.471} C_VEL
LIN {X 0,Y 516.491,Z 1000.006,A -85,B 0,C 180,E1 -5136.812,E2 -5136.812} C_VEL
LIN {X 0,Y 516.645,Z 993.206,A -85,B 0,C 180,E1 -5138.02,E2 -5138.02} C_VEL
LIN {X 0,Y 516.871,Z 984.957,A -85,B 0,C 180,E1 -5139.198,E2 -5139.198} C_VEL
LIN {X 0,Y 517.072,Z 976.496,A -85,B 0,C 180,E1 -5140.182,E2 -5140.182} C_VEL
LIN {X 0,Y 517.451,Z 966.038,A -85,B 0,C 180,E1 -5141.164,E2 -5141.164} C_VEL
LIN {X 0,Y 517.757,Z 954.682,A -85,B 0,C 180,E1 -5142.021,E2 -5142.021} C_VEL
LIN {X 0,Y 518.016,Z 942.401,A -85,B 0,C 180,E1 -5142.741,E2 -5142.741} C_VEL
LIN {X 0,Y 518.303,Z 930.06,A -85,B 0,C 180,E1 -5143.282,E2 -5143.282} C_VEL
LIN {X 0,Y 518.526,Z 917.358,A -85,B 0,C 180,E1 -5143.675,E2 -5143.675} C_VEL
LIN {X 0,Y 518.689,Z 904,A -85,B 0,C 180,E1 -5143.921,E2 -5143.921} C_VEL
LIN {X 0,Y 519.079,Z 812.576,A -85,B 0,C 180,E1 -5145.187,E2 -5145.187} C_VEL
LIN {X 0,Y 517.759,Z 801.542,A -85,B 0,C 180,E1 -5145.384,E2 -5145.384} C_VEL
LIN {X 0,Y 518.353,Z 773.664,A -85,B 0,C 180,E1 -5148.608,E2 -5148.608} C_VEL
LIN {X 0,Y 518.904,Z 749.337,A -85,B 0,C 180,E1 -5151.454,E2 -5151.454} C_VEL
LIN {X 0,Y 519.39,Z 728.256,A -85,B 0,C 180,E1 -5153.954,E2 -5153.954} C_VEL
LIN {X 0,Y 520.053,Z 702.446,A -85,B 0,C 180,E1 -5157.06,E2 -5157.06} C_VEL
LIN {X 0,Y 517.481,Z 690.801,A -85,B 0,C 180,E1 -5158.607,E2 -5158.607} C_VEL
LIN {X 0,Y 516.882,Z 688.103,A -85,B 0,C 180,E1 -5158.976,E2 -5158.976} C_VEL
LIN {X 0,Y 516.842,Z 688.101,A -85,B 0,C 180,E1 -5162.031,E2 -5162.031} C_VEL
LIN {X 0,Y 516.836,Z 688.108,A -85,B 0,C 180,E1 -5164.832,E2 -5164.832} C_VEL
LIN {X 0,Y 516.838,Z 688.102,A -85,B 0,C 180,E1 -5167.937,E2 -5167.937} C_VEL
LIN {X 0,Y 516.834,Z 688.105,A -85,B 0,C 180,E1 -5170.75,E2 -5170.75} C_VEL
LIN {X 0,Y 516.874,Z 688.097,A -85,B 0,C 180,E1 -5173.907,E2 -5173.907} C_VEL
LIN {X 0,Y 516.874,Z 688.096,A -85,B 0,C 180,E1 -5176.111,E2 -5176.111} C_VEL
LIN {X 0,Y 516.863,Z 688.106,A -85,B 0,C 180,E1 -5179.256,E2 -5179.256} C_VEL
LIN {X 0,Y 516.875,Z 688.096,A -85,B 0,C 180,E1 -5182.061,E2 -5182.061} C_VEL
LIN {X 0,Y 516.885,Z 688.102,A -85,B 0,C 180,E1 -5185.175,E2 -5185.175} C_VEL
LIN {X 0,Y 516.885,Z 688.096,A -85,B 0,C 180,E1 -5187.976,E2 -5187.976} C_VEL
LIN {X 0,Y 516.932,Z 688.091,A -85,B 0,C 180,E1 -5190.696,E2 -5190.696} C_VEL
LIN {X 0,Y 516.908,Z 688.096,A -85,B 0,C 180,E1 -5193.816,E2 -5193.816} C_VEL
LIN {X 0,Y 516.87,Z 688.099,A -85,B 0,C 180,E1 -5196.776,E2 -5196.776} C_VEL
LIN {X 0,Y 516.951,Z 688.093,A -85,B 0,C 180,E1 -5199.733,E2 -5199.733} C_VEL
LIN {X 0,Y 516.915,Z 688.094,A -85,B 0,C 180,E1 -5202.596,E2 -5202.596} C_VEL
LIN {X 0,Y 516.947,Z 688.096,A -85,B 0,C 180,E1 -5205.156,E2 -5205.156} C_VEL
LIN {X 0,Y 518.832,Z 694.284,A -85,B 0,C 180,E1 -5205.316,E2 -5205.316} C_VEL
LIN {X 0,Y 518.511,Z 766.668,A -85,B 0,C 180,E1 -5206.379,E2 -5206.379} C_VEL
LIN {X 0,Y 518.447,Z 778.378,A -85,B 0,C 180,E1 -5206.676,E2 -5206.676} C_VEL
LIN {X 0,Y 518.322,Z 789.19,A -85,B 0,C 180,E1 -5207.072,E2 -5207.072} C_VEL
LIN {X 0,Y 518.087,Z 799.268,A -85,B 0,C 180,E1 -5207.554,E2 -5207.554} C_VEL
LIN {X 0,Y 517.929,Z 809.11,A -85,B 0,C 180,E1 -5208.152,E2 -5208.152} C_VEL
LIN {X 0,Y 517.703,Z 817.253,A -85,B 0,C 180,E1 -5208.747,E2 -5208.747} C_VEL
LIN {X 0,Y 517.536,Z 825.182,A -85,B 0,C 180,E1 -5209.436,E2 -5209.436} C_VEL
LIN {X 0,Y 517.236,Z 834.442,A -85,B 0,C 180,E1 -5210.419,E2 -5210.419} C_VEL
LIN {X 0,Y 517.108,Z 840.69,A -85,B 0,C 180,E1 -5211.205,E2 -5211.205} C_VEL
LIN {X 0,Y 516.929,Z 847.226,A -85,B 0,C 180,E1 -5212.186,E2 -5212.186} C_VEL
LIN {X 0,Y 516.786,Z 852.417,A -85,B 0,C 180,E1 -5213.111,E2 -5213.111} C_VEL
LIN {X 0,Y 516.741,Z 857.173,A -85,B 0,C 180,E1 -5214.145,E2 -5214.145} C_VEL
LIN {X 0,Y 516.536,Z 861.461,A -85,B 0,C 180,E1 -5215.317,E2 -5215.317} C_VEL
LIN {X 0,Y 516.47,Z 865.433,A -85,B 0,C 180,E1 -5216.88,E2 -5216.88} C_VEL
LIN {X 0,Y 516.441,Z 866.912,A -85,B 0,C 180,E1 -5217.66,E2 -5217.66} C_VEL
LIN {X 0,Y 516.387,Z 868.471,A -85,B 0,C 180,E1 -5219.22,E2 -5219.22} C_VEL
LIN {X 0,Y 516.354,Z 868.688,A -85,B 0,C 180,E1 -5220,E2 -5220} C_VEL
LIN {X 0,Y 516.36,Z 868.485,A -85,B 0,C 180,E1 -5220.78,E2 -5220.78} C_VEL
LIN {X 0,Y 516.377,Z 866.905,A -85,B 0,C 180,E1 -5222.34,E2 -5222.34} C_VEL
LIN {X 0,Y 516.514,Z 863.688,A -85,B 0,C 180,E1 -5223.901,E2 -5223.901} C_VEL
LIN {X 0,Y 516.528,Z 860.154,A -85,B 0,C 180,E1 -5225.074,E2 -5225.074} C_VEL
LIN {X 0,Y 516.681,Z 855.498,A -85,B 0,C 180,E1 -5226.247,E2 -5226.247} C_VEL
LIN {X 0,Y 516.751,Z 850.729,A -85,B 0,C 180,E1 -5227.227,E2 -5227.227} C_VEL
LIN {X 0,Y 516.955,Z 843.586,A -85,B 0,C 180,E1 -5228.404,E2 -5228.404} C_VEL
LIN {X 0,Y 517.138,Z 836.326,A -85,B 0,C 180,E1 -5229.386,E2 -5229.386} C_VEL
LIN {X 0,Y 517.326,Z 829.453,A -85,B 0,C 180,E1 -5230.172,E2 -5230.172} C_VEL
LIN {X 0,Y 517.57,Z 821.298,A -85,B 0,C 180,E1 -5230.959,E2 -5230.959} C_VEL
LIN {X 0,Y 517.813,Z 811.372,A -85,B 0,C 180,E1 -5231.747,E2 -5231.747} C_VEL
LIN {X 0,Y 518.013,Z 802.119,A -85,B 0,C 180,E1 -5232.349,E2 -5232.349} C_VEL
LIN {X 0,Y 518.207,Z 791.959,A -85,B 0,C 180,E1 -5232.881,E2 -5232.881} C_VEL
LIN {X 0,Y 518.426,Z 781.658,A -85,B 0,C 180,E1 -5233.299,E2 -5233.299} C_VEL
LIN {X 0,Y 518.482,Z 770.91,A -85,B 0,C 180,E1 -5233.622,E2 -5233.622} C_VEL
LIN {X 0,Y 518.593,Z 758.16,A -85,B 0,C 180,E1 -5233.869,E2 -5233.869} C_VEL
LIN {X 0,Y 518.866,Z 694.118,A -85,B 0,C 180,E1 -5234.785,E2 -5234.785} C_VEL
LIN {X 0,Y 516.999,Z 688.088,A -85,B 0,C 180,E1 -5234.943,E2 -5234.943} C_VEL
LIN {X 0,Y 516.927,Z 688.093,A -85,B 0,C 180,E1 -5238.222,E2 -5238.222} C_VEL
LIN {X 0,Y 516.914,Z 688.1,A -85,B 0,C 180,E1 -5240.702,E2 -5240.702} C_VEL
LIN {X 0,Y 516.9,Z 688.093,A -85,B 0,C 180,E1 -5244.073,E2 -5244.073} C_VEL
LIN {X 0,Y 516.901,Z 688.099,A -85,B 0,C 180,E1 -5246.659,E2 -5246.659} C_VEL
LIN {X 0,Y 516.922,Z 688.091,A -85,B 0,C 180,E1 -5249.522,E2 -5249.522} C_VEL
LIN {X 0,Y 516.908,Z 688.095,A -85,B 0,C 180,E1 -5252.542,E2 -5252.542} C_VEL
LIN {X 0,Y 516.874,Z 688.099,A -85,B 0,C 180,E1 -5255.327,E2 -5255.327} C_VEL
LIN {X 0,Y 516.891,Z 688.093,A -85,B 0,C 180,E1 -5257.941,E2 -5257.941} C_VEL
LIN {X 0,Y 516.878,Z 688.098,A -85,B 0,C 180,E1 -5259.407,E2 -5259.407} C_VEL
LIN {X 0,Y 516.197,Z 688.181,A -85,B 0,C 180,E1 -5260.058,E2 -5260.058} C_VEL
LIN {X 0,Y 513.33,Z 688.543,A -85,B 0,C 180,E1 -5261.114,E2 -5261.114} C_VEL
LIN {X 0,Y 510.918,Z 688.84,A -85,B 0,C 180,E1 -5261.965,E2 -5261.965} C_VEL
LIN {X 0,Y 509.889,Z 688.968,A -85,B 0,C 180,E1 -5262.622,E2 -5262.622} C_VEL
LIN {X 0,Y 509.807,Z 688.98,A -85,B 0,C 180,E1 -5262.845,E2 -5262.845} C_VEL
LIN {X 0,Y 509.822,Z 688.973,A -85,B 0,C 180,E1 -5265.794,E2 -5265.794} C_VEL
LIN {X 0,Y 509.819,Z 688.975,A -85,B 0,C 180,E1 -5268.567,E2 -5268.567} C_VEL
LIN {X 0,Y 509.823,Z 688.974,A -85,B 0,C 180,E1 -5271.656,E2 -5271.656} C_VEL
LIN {X 0,Y 509.804,Z 688.977,A -85,B 0,C 180,E1 -5274.616,E2 -5274.616} C_VEL
LIN {X 0,Y 509.846,Z 688.975,A -85,B 0,C 180,E1 -5277.476,E2 -5277.476} C_VEL
LIN {X 0,Y 509.799,Z 688.976,A -85,B 0,C 180,E1 -5280.286,E2 -5280.286} C_VEL
LIN {X 0,Y 509.791,Z 688.981,A -85,B 0,C 180,E1 -5282.935,E2 -5282.935} C_VEL
LIN {X 0,Y 509.829,Z 688.979,A -85,B 0,C 180,E1 -5285.568,E2 -5285.568} C_VEL
LIN {X 0,Y 509.812,Z 688.977,A -85,B 0,C 180,E1 -5288.144,E2 -5288.144} C_VEL
LIN {X 0,Y 509.82,Z 688.977,A -85,B 0,C 180,E1 -5290.676,E2 -5290.676} C_VEL
LIN {X 0,Y 509.83,Z 688.982,A -85,B 0,C 180,E1 -5293.169,E2 -5293.169} C_VEL
LIN {X 0,Y 509.848,Z 688.976,A -85,B 0,C 180,E1 -5294.832,E2 -5294.832} C_VEL
LIN {X 0,Y 512.237,Z 696.165,A -85,B 0,C 180,E1 -5295.015,E2 -5295.015} C_VEL
LIN {X 0,Y 511.872,Z 769.442,A -85,B 0,C 180,E1 -5296.068,E2 -5296.068} C_VEL
LIN {X 0,Y 511.917,Z 782.598,A -85,B 0,C 180,E1 -5296.423,E2 -5296.423} C_VEL
LIN {X 0,Y 511.737,Z 795.536,A -85,B 0,C 180,E1 -5296.939,E2 -5296.939} C_VEL
LIN {X 0,Y 511.53,Z 807.424,A -85,B 0,C 180,E1 -5297.591,E2 -5297.591} C_VEL
LIN {X 0,Y 511.191,Z 818.818,A -85,B 0,C 180,E1 -5298.396,E2 -5298.396} C_VEL
LIN {X 0,Y 510.928,Z 828.948,A -85,B 0,C 180,E1 -5299.294,E2 -5299.294} C_VEL
LIN {X 0,Y 510.646,Z 838.025,A -85,B 0,C 180,E1 -5300.289,E2 -5300.289} C_VEL
LIN {X 0,Y 510.312,Z 846.814,A -85,B 0,C 180,E1 -5301.481,E2 -5301.481} C_VEL
LIN {X 0,Y 510.05,Z 854.499,A -85,B 0,C 180,E1 -5302.791,E2 -5302.791} C_VEL
LIN {X 0,Y 509.94,Z 860.295,A -85,B 0,C 180,E1 -5304.062,E2 -5304.062} C_VEL
LIN {X 0,Y 509.726,Z 864.549,A -85,B 0,C 180,E1 -5305.25,E2 -5305.25} C_VEL
LIN {X 0,Y 509.669,Z 866.787,A -85,B 0,C 180,E1 -5306.042,E2 -5306.042} C_VEL
LIN {X 0,Y 509.6,Z 868.614,A -85,B 0,C 180,E1 -5306.833,E2 -5306.833} C_VEL
LIN {X 0,Y 509.582,Z 869.992,A -85,B 0,C 180,E1 -5307.624,E2 -5307.624} C_VEL
LIN {X 0,Y 509.554,Z 871.575,A -85,B 0,C 180,E1 -5309.205,E2 -5309.205} C_VEL
LIN {X 0,Y 509.54,Z 871.812,A -85,B 0,C 180,E1 -5309.995,E2 -5309.995} C_VEL
LIN {X 0,Y 509.608,Z 871.064,A -85,B 0,C 180,E1 -5311.575,E2 -5311.575} C_VEL
LIN {X 0,Y 509.593,Z 868.818,A -85,B 0,C 180,E1 -5313.157,E2 -5313.157} C_VEL
LIN {X 0,Y 509.712,Z 866.016,A -85,B 0,C 180,E1 -5314.344,E2 -5314.344} C_VEL
LIN {X 0,Y 509.841,Z 862.218,A -85,B 0,C 180,E1 -5315.532,E2 -5315.532} C_VEL
LIN {X 0,Y 510.009,Z 856.768,A -85,B 0,C 180,E1 -5316.839,E2 -5316.839} C_VEL
LIN {X 0,Y 510.22,Z 849.943,A -85,B 0,C 180,E1 -5318.111,E2 -5318.111} C_VEL
LIN {X 0,Y 510.519,Z 841.937,A -85,B 0,C 180,E1 -5319.303,E2 -5319.303} C_VEL
LIN {X 0,Y 510.78,Z 833.733,A -85,B 0,C 180,E1 -5320.298,E2 -5320.298} C_VEL
LIN {X 0,Y 511.074,Z 823.585,A -85,B 0,C 180,E1 -5321.295,E2 -5321.295} C_VEL
LIN {X 0,Y 511.449,Z 813.144,A -85,B 0,C 180,E1 -5322.116,E2 -5322.116} C_VEL
LIN {X 0,Y 511.654,Z 801.912,A -85,B 0,C 180,E1 -5322.823,E2 -5322.823} C_VEL
LIN {X 0,Y 511.8,Z 790.081,A -85,B 0,C 180,E1 -5323.392,E2 -5323.392} C_VEL
LIN {X 0,Y 511.925,Z 776.761,A -85,B 0,C 180,E1 -5323.844,E2 -5323.844} C_VEL
LIN {X 0,Y 511.984,Z 763.572,A -85,B 0,C 180,E1 -5324.121,E2 -5324.121} C_VEL
LIN {X 0,Y 512.202,Z 695.79,A -85,B 0,C 180,E1 -5325.081,E2 -5325.081} C_VEL
LIN {X 0,Y 509.905,Z 688.971,A -85,B 0,C 180,E1 -5325.264,E2 -5325.264} C_VEL
LIN {X 0,Y 509.846,Z 688.979,A -85,B 0,C 180,E1 -5328.477,E2 -5328.477} C_VEL
LIN {X 0,Y 509.832,Z 688.982,A -85,B 0,C 180,E1 -5330.995,E2 -5330.995} C_VEL
LIN {X 0,Y 509.798,Z 688.978,A -85,B 0,C 180,E1 -5333.558,E2 -5333.558} C_VEL
LIN {X 0,Y 509.861,Z 688.968,A -85,B 0,C 180,E1 -5336.366,E2 -5336.366} C_VEL
LIN {X 0,Y 509.844,Z 688.974,A -85,B 0,C 180,E1 -5338.838,E2 -5338.838} C_VEL
LIN {X 0,Y 509.788,Z 688.983,A -85,B 0,C 180,E1 -5341.584,E2 -5341.584} C_VEL
LIN {X 0,Y 509.817,Z 688.974,A -85,B 0,C 180,E1 -5344.407,E2 -5344.407} C_VEL
LIN {X 0,Y 509.779,Z 688.985,A -85,B 0,C 180,E1 -5347.334,E2 -5347.334} C_VEL
LIN {X 0,Y 509.82,Z 688.975,A -85,B 0,C 180,E1 -5350.374,E2 -5350.374} C_VEL
LIN {X 0,Y 509.794,Z 688.98,A -85,B 0,C 180,E1 -5353.058,E2 -5353.058} C_VEL
LIN {X 0,Y 509.781,Z 688.981,A -85,B 0,C 180,E1 -5355.786,E2 -5355.786} C_VEL
LIN {X 0,Y 509.821,Z 688.975,A -85,B 0,C 180,E1 -5358.571,E2 -5358.571} C_VEL
LIN {X 0,Y 509.806,Z 688.981,A -85,B 0,C 180,E1 -5361.658,E2 -5361.658} C_VEL
LIN {X 0,Y 509.787,Z 688.978,A -85,B 0,C 180,E1 -5364.618,E2 -5364.618} C_VEL
LIN {X 0,Y 509.805,Z 688.977,A -85,B 0,C 180,E1 -5367.477,E2 -5367.477} C_VEL
LIN {X 0,Y 509.817,Z 688.978,A -85,B 0,C 180,E1 -5370.264,E2 -5370.264} C_VEL
LIN {X 0,Y 509.824,Z 688.974,A -85,B 0,C 180,E1 -5372.941,E2 -5372.941} C_VEL
LIN {X 0,Y 509.81,Z 688.975,A -85,B 0,C 180,E1 -5375.571,E2 -5375.571} C_VEL
LIN {X 0,Y 509.765,Z 688.985,A -85,B 0,C 180,E1 -5378.146,E2 -5378.146} C_VEL
LIN {X 0,Y 509.793,Z 688.981,A -85,B 0,C 180,E1 -5380.679,E2 -5380.679} C_VEL
LIN {X 0,Y 509.818,Z 688.973,A -85,B 0,C 180,E1 -5383.172,E2 -5383.172} C_VEL
LIN {X 0,Y 509.813,Z 688.975,A -85,B 0,C 180,E1 -5385.633,E2 -5385.633} C_VEL
LIN {X 0,Y 509.86,Z 688.972,A -85,B 0,C 180,E1 -5388.873,E2 -5388.873} C_VEL
LIN {X 0,Y 509.876,Z 688.969,A -85,B 0,C 180,E1 -5392.077,E2 -5392.077} C_VEL
LIN {X 0,Y 509.938,Z 688.964,A -85,B 0,C 180,E1 -5394.464,E2 -5394.464} C_VEL
LIN {X 0,Y 509.979,Z 688.955,A -85,B 0,C 180,E1 -5397.631,E2 -5397.631} C_VEL
LIN {X 0,Y 509.973,Z 688.956,A -85,B 0,C 180,E1 -5400,E2 -5400} C_VEL
LIN {X 0,Y 509.917,Z 688.968,A -85,B 0,C 180,E1 -5403.16,E2 -5403.16} C_VEL
LIN {X 0,Y 509.905,Z 688.965,A -85,B 0,C 180,E1 -5406.331,E2 -5406.331} C_VEL
LIN {X 0,Y 509.875,Z 688.968,A -85,B 0,C 180,E1 -5408.721,E2 -5408.721} C_VEL
LIN {X 0,Y 509.874,Z 688.97,A -85,B 0,C 180,E1 -5411.932,E2 -5411.932} C_VEL
LIN {X 0,Y 509.827,Z 688.98,A -85,B 0,C 180,E1 -5415.248,E2 -5415.248} C_VEL
LIN {X 0,Y 509.815,Z 688.977,A -85,B 0,C 180,E1 -5418.004,E2 -5418.004} C_VEL
LIN {X 0,Y 509.785,Z 688.976,A -85,B 0,C 180,E1 -5421.005,E2 -5421.005} C_VEL
LIN {X 0,Y 509.792,Z 688.985,A -85,B 0,C 180,E1 -5423.565,E2 -5423.565} C_VEL
LIN {X 0,Y 509.851,Z 688.97,A -85,B 0,C 180,E1 -5426.384,E2 -5426.384} C_VEL
LIN {X 0,Y 509.82,Z 688.974,A -85,B 0,C 180,E1 -5428.848,E2 -5428.848} C_VEL
LIN {X 0,Y 509.77,Z 688.983,A -85,B 0,C 180,E1 -5431.594,E2 -5431.594} C_VEL
LIN {X 0,Y 509.794,Z 688.981,A -85,B 0,C 180,E1 -5434.418,E2 -5434.418} C_VEL
LIN {X 0,Y 509.763,Z 688.981,A -85,B 0,C 180,E1 -5437.346,E2 -5437.346} C_VEL
LIN {X 0,Y 509.828,Z 688.981,A -85,B 0,C 180,E1 -5440.383,E2 -5440.383} C_VEL
LIN {X 0,Y 509.79,Z 688.979,A -85,B 0,C 180,E1 -5443.07,E2 -5443.07} C_VEL
LIN {X 0,Y 509.782,Z 688.981,A -85,B 0,C 180,E1 -5445.798,E2 -5445.798} C_VEL
LIN {X 0,Y 509.827,Z 688.982,A -85,B 0,C 180,E1 -5448.582,E2 -5448.582} C_VEL
LIN {X 0,Y 509.811,Z 688.977,A -85,B 0,C 180,E1 -5451.793,E2 -5451.793} C_VEL
LIN {X 0,Y 509.807,Z 688.984,A -85,B 0,C 180,E1 -5454.629,E2 -5454.629} C_VEL
LIN {X 0,Y 509.828,Z 688.977,A -85,B 0,C 180,E1 -5457.487,E2 -5457.487} C_VEL
LIN {X 0,Y 509.86,Z 689.011,A -85,B 0,C 180,E1 -5460.824,E2 -5460.824} C_VEL
LIN {X 0,Y 513.059,Z 703.351,A -85,B 0,C 180,E1 -5462.773,E2 -5462.773} C_VEL
LIN {X 0,Y 512.682,Z 722.147,A -85,B 0,C 180,E1 -5465.076,E2 -5465.076} C_VEL
LIN {X 0,Y 511.948,Z 748.514,A -85,B 0,C 180,E1 -5468.251,E2 -5468.251} C_VEL
LIN {X 0,Y 511.269,Z 776.533,A -85,B 0,C 180,E1 -5471.576,E2 -5471.576} C_VEL
LIN {X 0,Y 510.752,Z 800.852,A -85,B 0,C 180,E1 -5474.41,E2 -5474.41} C_VEL
LIN {X 0,Y 512.217,Z 813.607,A -85,B 0,C 180,E1 -5474.634,E2 -5474.634} C_VEL
LIN {X 0,Y 511.717,Z 911.379,A -85,B 0,C 180,E1 -5476.023,E2 -5476.023} C_VEL
LIN {X 0,Y 511.447,Z 924.636,A -85,B 0,C 180,E1 -5476.37,E2 -5476.37} C_VEL
LIN {X 0,Y 511.162,Z 936.861,A -85,B 0,C 180,E1 -5476.843,E2 -5476.843} C_VEL
LIN {X 0,Y 510.924,Z 949.313,A -85,B 0,C 180,E1 -5477.497,E2 -5477.497} C_VEL
LIN {X 0,Y 510.591,Z 961.001,A -85,B 0,C 180,E1 -5478.292,E2 -5478.292} C_VEL
LIN {X 0,Y 510.238,Z 971.578,A -85,B 0,C 180,E1 -5479.189,E2 -5479.189} C_VEL
LIN {X 0,Y 510.027,Z 980.161,A -85,B 0,C 180,E1 -5480.088,E2 -5480.088} C_VEL
LIN {X 0,Y 509.757,Z 988.003,A -85,B 0,C 180,E1 -5481.083,E2 -5481.083} C_VEL
LIN {X 0,Y 509.525,Z 995.654,A -85,B 0,C 180,E1 -5482.277,E2 -5482.277} C_VEL
LIN {X 0,Y 509.335,Z 1002.704,A -85,B 0,C 180,E1 -5483.668,E2 -5483.668} C_VEL
LIN {X 0,Y 509.245,Z 1007.392,A -85,B 0,C 180,E1 -5484.859,E2 -5484.859} C_VEL
LIN {X 0,Y 509.252,Z 1010.975,A -85,B 0,C 180,E1 -5486.049,E2 -5486.049} C_VEL
LIN {X 0,Y 509.199,Z 1012.821,A -85,B 0,C 180,E1 -5486.841,E2 -5486.841} C_VEL
LIN {X 0,Y 509.16,Z 1014.203,A -85,B 0,C 180,E1 -5487.632,E2 -5487.632} C_VEL
LIN {X 0,Y 509.073,Z 1015.789,A -85,B 0,C 180,E1 -5489.214,E2 -5489.214} C_VEL
LIN {X 0,Y 509.065,Z 1016,A -85,B 0,C 180,E1 -5490.005,E2 -5490.005} C_VEL
LIN {X 0,Y 509.112,Z 1015.176,A -85,B 0,C 180,E1 -5491.587,E2 -5491.587} C_VEL
LIN {X 0,Y 509.161,Z 1014.186,A -85,B 0,C 180,E1 -5492.378,E2 -5492.378} C_VEL
LIN {X 0,Y 509.202,Z 1012.796,A -85,B 0,C 180,E1 -5493.17,E2 -5493.17} C_VEL
LIN {X 0,Y 509.235,Z 1009.88,A -85,B 0,C 180,E1 -5494.358,E2 -5494.358} C_VEL
LIN {X 0,Y 509.347,Z 1005.932,A -85,B 0,C 180,E1 -5495.548,E2 -5495.548} C_VEL
LIN {X 0,Y 509.415,Z 1000.257,A -85,B 0,C 180,E1 -5496.858,E2 -5496.858} C_VEL
LIN {X 0,Y 509.589,Z 993.205,A -85,B 0,C 180,E1 -5498.131,E2 -5498.131} C_VEL
LIN {X 0,Y 509.85,Z 984.957,A -85,B 0,C 180,E1 -5499.326,E2 -5499.326} C_VEL
LIN {X 0,Y 510.061,Z 976.463,A -85,B 0,C 180,E1 -5500.323,E2 -5500.323} C_VEL
LIN {X 0,Y 510.466,Z 965.857,A -85,B 0,C 180,E1 -5501.319,E2 -5501.319} C_VEL
LIN {X 0,Y 510.803,Z 954.177,A -85,B 0,C 180,E1 -5502.196,E2 -5502.196} C_VEL
LIN {X 0,Y 511.067,Z 941.828,A -85,B 0,C 180,E1 -5502.917,E2 -5502.917} C_VEL
LIN {X 0,Y 511.343,Z 929.344,A -85,B 0,C 180,E1 -5503.466,E2 -5503.466} C_VEL
LIN {X 0,Y 511.626,Z 916.538,A -85,B 0,C 180,E1 -5503.863,E2 -5503.863} C_VEL
LIN {X 0,Y 511.782,Z 903.099,A -85,B 0,C 180,E1 -5504.112,E2 -5504.112} C_VEL
LIN {X 0,Y 512.151,Z 811.846,A -85,B 0,C 180,E1 -5505.393,E2 -5505.393} C_VEL
LIN {X 0,Y 510.742,Z 800.522,A -85,B 0,C 180,E1 -5505.601,E2 -5505.601} C_VEL
LIN {X 0,Y 511.312,Z 774.818,A -85,B 0,C 180,E1 -5508.62,E2 -5508.62} C_VEL
LIN {X 0,Y 511.923,Z 750.175,A -85,B 0,C 180,E1 -5511.549,E2 -5511.549} C_VEL
LIN {X 0,Y 512.461,Z 729.108,A -85,B 0,C 180,E1 -5514.083,E2 -5514.083} C_VEL
LIN {X 0,Y 513.164,Z 703.756,A -85,B 0,C 180,E1 -5517.174,E2 -5517.174} C_VEL
LIN {X 0,Y 509.828,Z 688.982,A -85,B 0,C 180,E1 -5519.19,E2 -5519.19} C_VEL
LIN {X 0,Y 509.829,Z 688.975,A -85,B 0,C 180,E1 -5522.525,E2 -5522.525} C_VEL
LIN {X 0,Y 509.774,Z 688.979,A -85,B 0,C 180,E1 -5525.57,E2 -5525.57} C_VEL
LIN {X 0,Y 509.809,Z 688.977,A -85,B 0,C 180,E1 -5528.345,E2 -5528.345} C_VEL
LIN {X 0,Y 509.797,Z 688.983,A -85,B 0,C 180,E1 -5531.435,E2 -5531.435} C_VEL
LIN {X 0,Y 509.85,Z 688.973,A -85,B 0,C 180,E1 -5534.672,E2 -5534.672} C_VEL
LIN {X 0,Y 509.803,Z 688.982,A -85,B 0,C 180,E1 -5537.507,E2 -5537.507} C_VEL
LIN {X 0,Y 509.844,Z 688.974,A -85,B 0,C 180,E1 -5540.647,E2 -5540.647} C_VEL
LIN {X 0,Y 509.811,Z 688.98,A -85,B 0,C 180,E1 -5543.646,E2 -5543.646} C_VEL
LIN {X 0,Y 509.852,Z 688.971,A -85,B 0,C 180,E1 -5546.538,E2 -5546.538} C_VEL
LIN {X 0,Y 509.853,Z 688.979,A -85,B 0,C 180,E1 -5549.335,E2 -5549.335} C_VEL
LIN {X 0,Y 509.851,Z 688.973,A -85,B 0,C 180,E1 -5552.052,E2 -5552.052} C_VEL
LIN {X 0,Y 509.826,Z 688.977,A -85,B 0,C 180,E1 -5554.701,E2 -5554.701} C_VEL
LIN {X 0,Y 509.838,Z 688.98,A -85,B 0,C 180,E1 -5557.459,E2 -5557.459} C_VEL
LIN {X 0,Y 509.928,Z 688.967,A -85,B 0,C 180,E1 -5559.845,E2 -5559.845} C_VEL
LIN {X 0,Y 509.879,Z 688.975,A -85,B 0,C 180,E1 -5563.175,E2 -5563.175} C_VEL
LIN {X 0,Y 509.914,Z 688.97,A -85,B 0,C 180,E1 -5564.97,E2 -5564.97} C_VEL
LIN {X 0,Y 512.038,Z 696.121,A -85,B 0,C 180,E1 -5565.147,E2 -5565.147} C_VEL
LIN {X 0,Y 511.616,Z 767.588,A -85,B 0,C 180,E1 -5566.217,E2 -5566.217} C_VEL
LIN {X 0,Y 511.557,Z 779.363,A -85,B 0,C 180,E1 -5566.519,E2 -5566.519} C_VEL
LIN {X 0,Y 511.426,Z 789.661,A -85,B 0,C 180,E1 -5566.895,E2 -5566.895} C_VEL
LIN {X 0,Y 511.209,Z 799.96,A -85,B 0,C 180,E1 -5567.388,E2 -5567.388} C_VEL
LIN {X 0,Y 511.028,Z 809.911,A -85,B 0,C 180,E1 -5567.994,E2 -5567.994} C_VEL
LIN {X 0,Y 510.773,Z 819.232,A -85,B 0,C 180,E1 -5568.693,E2 -5568.693} C_VEL
LIN {X 0,Y 510.61,Z 826.05,A -85,B 0,C 180,E1 -5569.291,E2 -5569.291} C_VEL
LIN {X 0,Y 510.299,Z 835.363,A -85,B 0,C 180,E1 -5570.287,E2 -5570.287} C_VEL
LIN {X 0,Y 510.164,Z 841.645,A -85,B 0,C 180,E1 -5571.084,E2 -5571.084} C_VEL
LIN {X 0,Y 509.971,Z 848.212,A -85,B 0,C 180,E1 -5572.079,E2 -5572.079} C_VEL
LIN {X 0,Y 509.811,Z 853.417,A -85,B 0,C 180,E1 -5573.015,E2 -5573.015} C_VEL
LIN {X 0,Y 509.762,Z 858.192,A -85,B 0,C 180,E1 -5574.065,E2 -5574.065} C_VEL
LIN {X 0,Y 509.535,Z 862.497,A -85,B 0,C 180,E1 -5575.253,E2 -5575.253} C_VEL
LIN {X 0,Y 509.458,Z 866.477,A -85,B 0,C 180,E1 -5576.837,E2 -5576.837} C_VEL
LIN {X 0,Y 509.443,Z 867.955,A -85,B 0,C 180,E1 -5577.628,E2 -5577.628} C_VEL
LIN {X 0,Y 509.389,Z 869.505,A -85,B 0,C 180,E1 -5579.21,E2 -5579.21} C_VEL
LIN {X 0,Y 509.356,Z 869.716,A -85,B 0,C 180,E1 -5580,E2 -5580} C_VEL
LIN {X 0,Y 509.339,Z 869.509,A -85,B 0,C 180,E1 -5580.791,E2 -5580.791} C_VEL
LIN {X 0,Y 509.354,Z 867.905,A -85,B 0,C 180,E1 -5582.372,E2 -5582.372} C_VEL
LIN {X 0,Y 509.497,Z 864.656,A -85,B 0,C 180,E1 -5583.955,E2 -5583.955} C_VEL
LIN {X 0,Y 509.528,Z 861.092,A -85,B 0,C 180,E1 -5585.144,E2 -5585.144} C_VEL
LIN {X 0,Y 509.695,Z 856.401,A -85,B 0,C 180,E1 -5586.333,E2 -5586.333} C_VEL
LIN {X 0,Y 509.771,Z 851.596,A -85,B 0,C 180,E1 -5587.327,E2 -5587.327} C_VEL
LIN {X 0,Y 509.992,Z 844.41,A -85,B 0,C 180,E1 -5588.519,E2 -5588.519} C_VEL
LIN {X 0,Y 510.182,Z 837.1,A -85,B 0,C 180,E1 -5589.515,E2 -5589.515} C_VEL
LIN {X 0,Y 510.385,Z 830.177,A -85,B 0,C 180,E1 -5590.312,E2 -5590.312} C_VEL
LIN {X 0,Y 510.642,Z 821.961,A -85,B 0,C 180,E1 -5591.109,E2 -5591.109} C_VEL
LIN {X 0,Y 510.845,Z 813.388,A -85,B 0,C 180,E1 -5591.809,E2 -5591.809} C_VEL
LIN {X 0,Y 511.096,Z 803.115,A -85,B 0,C 180,E1 -5592.49,E2 -5592.49} C_VEL
LIN {X 0,Y 511.31,Z 792.324,A -85,B 0,C 180,E1 -5593.058,E2 -5593.058} C_VEL
LIN {X 0,Y 511.503,Z 782.588,A -85,B 0,C 180,E1 -5593.457,E2 -5593.457} C_VEL
LIN {X 0,Y 511.576,Z 771.858,A -85,B 0,C 180,E1 -5593.784,E2 -5593.784} C_VEL
LIN {X 0,Y 511.693,Z 759.163,A -85,B 0,C 180,E1 -5594.035,E2 -5594.035} C_VEL
LIN {X 0,Y 511.939,Z 695.318,A -85,B 0,C 180,E1 -5594.969,E2 -5594.969} C_VEL
LIN {X 0,Y 509.931,Z 688.967,A -85,B 0,C 180,E1 -5595.136,E2 -5595.136} C_VEL
LIN {X 0,Y 509.872,Z 688.975,A -85,B 0,C 180,E1 -5598.483,E2 -5598.483} C_VEL
LIN {X 0,Y 509.856,Z 688.975,A -85,B 0,C 180,E1 -5601.002,E2 -5601.002} C_VEL
LIN {X 0,Y 509.833,Z 688.973,A -85,B 0,C 180,E1 -5603.563,E2 -5603.563} C_VEL
LIN {X 0,Y 509.866,Z 688.971,A -85,B 0,C 180,E1 -5606.364,E2 -5606.364} C_VEL
LIN {X 0,Y 509.863,Z 688.978,A -85,B 0,C 180,E1 -5608.845,E2 -5608.845} C_VEL
LIN {X 0,Y 509.832,Z 688.974,A -85,B 0,C 180,E1 -5611.59,E2 -5611.59} C_VEL
LIN {X 0,Y 509.848,Z 688.972,A -85,B 0,C 180,E1 -5614.414,E2 -5614.414} C_VEL
LIN {X 0,Y 509.822,Z 688.977,A -85,B 0,C 180,E1 -5617.341,E2 -5617.341} C_VEL
LIN {X 0,Y 509.829,Z 688.974,A -85,B 0,C 180,E1 -5620.383,E2 -5620.383} C_VEL
LIN {X 0,Y 509.807,Z 688.98,A -85,B 0,C 180,E1 -5622.845,E2 -5622.845} C_VEL
LIN {X 0,Y 509.145,Z 689.067,A -85,B 0,C 180,E1 -5623.504,E2 -5623.504} C_VEL
LIN {X 0,Y 506.284,Z 689.42,A -85,B 0,C 180,E1 -5624.574,E2 -5624.574} C_VEL
LIN {X 0,Y 503.864,Z 689.718,A -85,B 0,C 180,E1 -5625.436,E2 -5625.436} C_VEL
LIN {X 0,Y 502.83,Z 689.844,A -85,B 0,C 180,E1 -5626.102,E2 -5626.102} C_VEL
LIN {X 0,Y 502.749,Z 689.854,A -85,B 0,C 180,E1 -5626.327,E2 -5626.327} C_VEL
LIN {X 0,Y 502.779,Z 689.857,A -85,B 0,C 180,E1 -5629.011,E2 -5629.011} C_VEL
LIN {X 0,Y 502.77,Z 689.851,A -85,B 0,C 180,E1 -5632.04,E2 -5632.04} C_VEL
LIN {X 0,Y 502.783,Z 689.857,A -85,B 0,C 180,E1 -5635.029,E2 -5635.029} C_VEL
LIN {X 0,Y 502.771,Z 689.852,A -85,B 0,C 180,E1 -5637.911,E2 -5637.911} C_VEL
LIN {X 0,Y 502.764,Z 689.854,A -85,B 0,C 180,E1 -5640.705,E2 -5640.705} C_VEL
LIN {X 0,Y 502.75,Z 689.861,A -85,B 0,C 180,E1 -5643.466,E2 -5643.466} C_VEL
LIN {X 0,Y 502.764,Z 689.855,A -85,B 0,C 180,E1 -5646.081,E2 -5646.081} C_VEL
LIN {X 0,Y 502.767,Z 689.856,A -85,B 0,C 180,E1 -5648.684,E2 -5648.684} C_VEL
LIN {X 0,Y 502.801,Z 689.854,A -85,B 0,C 180,E1 -5651.895,E2 -5651.895} C_VEL
LIN {X 0,Y 502.826,Z 690.03,A -85,B 0,C 180,E1 -5654.618,E2 -5654.618} C_VEL
LIN {X 0,Y 505.387,Z 697.499,A -85,B 0,C 180,E1 -5654.812,E2 -5654.812} C_VEL
LIN {X 0,Y 505.031,Z 770.471,A -85,B 0,C 180,E1 -5655.875,E2 -5655.875} C_VEL
LIN {X 0,Y 505.072,Z 783.619,A -85,B 0,C 180,E1 -5656.235,E2 -5656.235} C_VEL
LIN {X 0,Y 504.892,Z 796.551,A -85,B 0,C 180,E1 -5656.758,E2 -5656.758} C_VEL
LIN {X 0,Y 504.67,Z 808.425,A -85,B 0,C 180,E1 -5657.419,E2 -5657.419} C_VEL
LIN {X 0,Y 504.313,Z 819.827,A -85,B 0,C 180,E1 -5658.236,E2 -5658.236} C_VEL
LIN {X 0,Y 504.029,Z 829.956,A -85,B 0,C 180,E1 -5659.145,E2 -5659.145} C_VEL
LIN {X 0,Y 503.729,Z 839.031,A -85,B 0,C 180,E1 -5660.155,E2 -5660.155} C_VEL
LIN {X 0,Y 503.367,Z 847.82,A -85,B 0,C 180,E1 -5661.363,E2 -5661.363} C_VEL
LIN {X 0,Y 503.079,Z 855.505,A -85,B 0,C 180,E1 -5662.691,E2 -5662.691} C_VEL
LIN {X 0,Y 502.962,Z 861.298,A -85,B 0,C 180,E1 -5663.979,E2 -5663.979} C_VEL
LIN {X 0,Y 502.723,Z 865.554,A -85,B 0,C 180,E1 -5665.183,E2 -5665.183} C_VEL
LIN {X 0,Y 502.657,Z 867.791,A -85,B 0,C 180,E1 -5665.986,E2 -5665.986} C_VEL
LIN {X 0,Y 502.583,Z 869.618,A -85,B 0,C 180,E1 -5666.788,E2 -5666.788} C_VEL
LIN {X 0,Y 502.571,Z 870.994,A -85,B 0,C 180,E1 -5667.59,E2 -5667.59} C_VEL
LIN {X 0,Y 502.539,Z 872.577,A -85,B 0,C 180,E1 -5669.193,E2 -5669.193} C_VEL
LIN {X 0,Y 502.523,Z 872.813,A -85,B 0,C 180,E1 -5669.995,E2 -5669.995} C_VEL
LIN {X 0,Y 502.599,Z 872.064,A -85,B 0,C 180,E1 -5671.597,E2 -5671.597} C_VEL
LIN {X 0,Y 502.575,Z 869.82,A -85,B 0,C 180,E1 -5673.201,E2 -5673.201} C_VEL
LIN {X 0,Y 502.705,Z 867.018,A -85,B 0,C 180,E1 -5674.404,E2 -5674.404} C_VEL
LIN {X 0,Y 502.858,Z 863.216,A -85,B 0,C 180,E1 -5675.609,E2 -5675.609} C_VEL
LIN {X 0,Y 503.033,Z 857.757,A -85,B 0,C 180,E1 -5676.936,E2 -5676.936} C_VEL
LIN {X 0,Y 503.265,Z 850.942,A -85,B 0,C 180,E1 -5678.224,E2 -5678.224} C_VEL
LIN {X 0,Y 503.585,Z 842.935,A -85,B 0,C 180,E1 -5679.432,E2 -5679.432} C_VEL
LIN {X 0,Y 503.873,Z 834.73,A -85,B 0,C 180,E1 -5680.441,E2 -5680.441} C_VEL
LIN {X 0,Y 504.184,Z 824.581,A -85,B 0,C 180,E1 -5681.451,E2 -5681.451} C_VEL
LIN {X 0,Y 504.581,Z 814.139,A -85,B 0,C 180,E1 -5682.283,E2 -5682.283} C_VEL
LIN {X 0,Y 504.819,Z 802.385,A -85,B 0,C 180,E1 -5683.03,E2 -5683.03} C_VEL
LIN {X 0,Y 504.973,Z 789.91,A -85,B 0,C 180,E1 -5683.623,E2 -5683.623} C_VEL
LIN {X 0,Y 505.104,Z 776.838,A -85,B 0,C 180,E1 -5684.061,E2 -5684.061} C_VEL
LIN {X 0,Y 505.145,Z 764.545,A -85,B 0,C 180,E1 -5684.317,E2 -5684.317} C_VEL
LIN {X 0,Y 505.388,Z 697.338,A -85,B 0,C 180,E1 -5685.281,E2 -5685.281} C_VEL
LIN {X 0,Y 502.829,Z 689.851,A -85,B 0,C 180,E1 -5685.499,E2 -5685.499} C_VEL
LIN {X 0,Y 502.81,Z 689.857,A -85,B 0,C 180,E1 -5688.746,E2 -5688.746} C_VEL
LIN {X 0,Y 502.764,Z 689.857,A -85,B 0,C 180,E1 -5691.305,E2 -5691.305} C_VEL
LIN {X 0,Y 502.747,Z 689.855,A -85,B 0,C 180,E1 -5693.908,E2 -5693.908} C_VEL
LIN {X 0,Y 502.811,Z 689.847,A -85,B 0,C 180,E1 -5696.561,E2 -5696.561} C_VEL
LIN {X 0,Y 502.793,Z 689.856,A -85,B 0,C 180,E1 -5699.281,E2 -5699.281} C_VEL
LIN {X 0,Y 502.751,Z 689.856,A -85,B 0,C 180,E1 -5702.078,E2 -5702.078} C_VEL
LIN {X 0,Y 502.772,Z 689.855,A -85,B 0,C 180,E1 -5704.959,E2 -5704.959} C_VEL
LIN {X 0,Y 502.754,Z 689.85,A -85,B 0,C 180,E1 -5707.948,E2 -5707.948} C_VEL
LIN {X 0,Y 502.786,Z 689.854,A -85,B 0,C 180,E1 -5711.059,E2 -5711.059} C_VEL
LIN {X 0,Y 502.737,Z 689.863,A -85,B 0,C 180,E1 -5713.37,E2 -5713.37} C_VEL
LIN {X 0,Y 502.741,Z 689.856,A -85,B 0,C 180,E1 -5715.655,E2 -5715.655} C_VEL
LIN {X 0,Y 502.787,Z 689.859,A -85,B 0,C 180,E1 -5717.859,E2 -5717.859} C_VEL
LIN {X 0,Y 502.776,Z 689.851,A -85,B 0,C 180,E1 -5721.021,E2 -5721.021} C_VEL
LIN {X 0,Y 502.727,Z 689.863,A -85,B 0,C 180,E1 -5724.162,E2 -5724.162} C_VEL
LIN {X 0,Y 502.772,Z 689.851,A -85,B 0,C 180,E1 -5726.988,E2 -5726.988} C_VEL
LIN {X 0,Y 502.768,Z 689.859,A -85,B 0,C 180,E1 -5730.057,E2 -5730.057} C_VEL
LIN {X 0,Y 502.771,Z 689.856,A -85,B 0,C 180,E1 -5732.529,E2 -5732.529} C_VEL
LIN {X 0,Y 502.764,Z 689.852,A -85,B 0,C 180,E1 -5735.293,E2 -5735.293} C_VEL
LIN {X 0,Y 502.733,Z 689.857,A -85,B 0,C 180,E1 -5737.824,E2 -5737.824} C_VEL
LIN {X 0,Y 502.754,Z 689.863,A -85,B 0,C 180,E1 -5740.397,E2 -5740.397} C_VEL
LIN {X 0,Y 502.766,Z 689.853,A -85,B 0,C 180,E1 -5742.929,E2 -5742.929} C_VEL
LIN {X 0,Y 502.791,Z 689.85,A -85,B 0,C 180,E1 -5745.427,E2 -5745.427} C_VEL
LIN {X 0,Y 502.826,Z 689.849,A -85,B 0,C 180,E1 -5748.716,E2 -5748.716} C_VEL
LIN {X 0,Y 502.83,Z 689.846,A -85,B 0,C 180,E1 -5751.965,E2 -5751.965} C_VEL
LIN {X 0,Y 502.889,Z 689.841,A -85,B 0,C 180,E1 -5754.386,E2 -5754.386} C_VEL
LIN {X 0,Y 502.951,Z 689.831,A -85,B 0,C 180,E1 -5757.597,E2 -5757.597} C_VEL
LIN {X 0,Y 502.945,Z 689.832,A -85,B 0,C 180,E1 -5760,E2 -5760} C_VEL
LIN {X 0,Y 502.951,Z 689.829,A -85,B 0,C 180,E1 -5762.403,E2 -5762.403} C_VEL
LIN {X 0,Y 502.889,Z 689.842,A -85,B 0,C 180,E1 -5765.614,E2 -5765.614} C_VEL
LIN {X 0,Y 502.826,Z 689.847,A -85,B 0,C 180,E1 -5768.844,E2 -5768.844} C_VEL
LIN {X 0,Y 502.819,Z 689.847,A -85,B 0,C 180,E1 -5772.102,E2 -5772.102} C_VEL
LIN {X 0,Y 502.776,Z 689.861,A -85,B 0,C 180,E1 -5775.402,E2 -5775.402} C_VEL
LIN {X 0,Y 502.773,Z 689.854,A -85,B 0,C 180,E1 -5778.126,E2 -5778.126} C_VEL
LIN {X 0,Y 502.725,Z 689.859,A -85,B 0,C 180,E1 -5781.314,E2 -5781.314} C_VEL
LIN {X 0,Y 502.751,Z 689.86,A -85,B 0,C 180,E1 -5783.916,E2 -5783.916} C_VEL
LIN {X 0,Y 502.813,Z 689.846,A -85,B 0,C 180,E1 -5786.569,E2 -5786.569} C_VEL
LIN {X 0,Y 502.774,Z 689.853,A -85,B 0,C 180,E1 -5789.291,E2 -5789.291} C_VEL
LIN {X 0,Y 502.728,Z 689.865,A -85,B 0,C 180,E1 -5792.089,E2 -5792.089} C_VEL
LIN {X 0,Y 502.75,Z 689.855,A -85,B 0,C 180,E1 -5794.97,E2 -5794.97} C_VEL
LIN {X 0,Y 502.742,Z 689.861,A -85,B 0,C 180,E1 -5797.959,E2 -5797.959} C_VEL
LIN {X 0,Y 502.779,Z 689.852,A -85,B 0,C 180,E1 -5801.002,E2 -5801.002} C_VEL
LIN {X 0,Y 502.732,Z 689.858,A -85,B 0,C 180,E1 -5803.381,E2 -5803.381} C_VEL
LIN {X 0,Y 502.742,Z 689.857,A -85,B 0,C 180,E1 -5805.667,E2 -5805.667} C_VEL
LIN {X 0,Y 502.793,Z 689.849,A -85,B 0,C 180,E1 -5807.871,E2 -5807.871} C_VEL
LIN {X 0,Y 502.768,Z 689.856,A -85,B 0,C 180,E1 -5811.031,E2 -5811.031} C_VEL
LIN {X 0,Y 502.745,Z 689.859,A -85,B 0,C 180,E1 -5814.174,E2 -5814.174} C_VEL
LIN {X 0,Y 502.799,Z 689.852,A -85,B 0,C 180,E1 -5817,E2 -5817} C_VEL
LIN {X 0,Y 502.809,Z 689.857,A -85,B 0,C 180,E1 -5820.515,E2 -5820.515} C_VEL
LIN {X 0,Y 502.821,Z 689.961,A -85,B 0,C 180,E1 -5820.618,E2 -5820.618} C_VEL
LIN {X 0,Y 506.195,Z 705.327,A -85,B 0,C 180,E1 -5822.739,E2 -5822.739} C_VEL
LIN {X 0,Y 505.747,Z 723.072,A -85,B 0,C 180,E1 -5824.941,E2 -5824.941} C_VEL
LIN {X 0,Y 505.095,Z 745.847,A -85,B 0,C 180,E1 -5827.726,E2 -5827.726} C_VEL
LIN {X 0,Y 504.341,Z 772.047,A -85,B 0,C 180,E1 -5830.892,E2 -5830.892} C_VEL
LIN {X 0,Y 503.829,Z 792.944,A -85,B 0,C 180,E1 -5833.391,E2 -5833.391} C_VEL
LIN {X 0,Y 503.687,Z 799.488,A -85,B 0,C 180,E1 -5834.172,E2 -5834.172} C_VEL
LIN {X 0,Y 505.347,Z 814.476,A -85,B 0,C 180,E1 -5834.447,E2 -5834.447} C_VEL
LIN {X 0,Y 504.822,Z 910.365,A -85,B 0,C 180,E1 -5835.828,E2 -5835.828} C_VEL
LIN {X 0,Y 504.51,Z 923.617,A -85,B 0,C 180,E1 -5836.179,E2 -5836.179} C_VEL
LIN {X 0,Y 504.184,Z 936.972,A -85,B 0,C 180,E1 -5836.709,E2 -5836.709} C_VEL
LIN {X 0,Y 503.91,Z 948.776,A -85,B 0,C 180,E1 -5837.351,E2 -5837.351} C_VEL
LIN {X 0,Y 503.603,Z 959.982,A -85,B 0,C 180,E1 -5838.127,E2 -5838.127} C_VEL
LIN {X 0,Y 503.233,Z 970.57,A -85,B 0,C 180,E1 -5839.037,E2 -5839.037} C_VEL
LIN {X 0,Y 502.957,Z 979.256,A -85,B 0,C 180,E1 -5839.947,E2 -5839.947} C_VEL
LIN {X 0,Y 502.695,Z 987.282,A -85,B 0,C 180,E1 -5840.957,E2 -5840.957} C_VEL
LIN {X 0,Y 502.443,Z 995.139,A -85,B 0,C 180,E1 -5842.168,E2 -5842.168} C_VEL
LIN {X 0,Y 502.269,Z 1002.394,A -85,B 0,C 180,E1 -5843.579,E2 -5843.579} C_VEL
LIN {X 0,Y 502.183,Z 1007.226,A -85,B 0,C 180,E1 -5844.786,E2 -5844.786} C_VEL
LIN {X 0,Y 502.148,Z 1010.895,A -85,B 0,C 180,E1 -5845.993,E2 -5845.993} C_VEL
LIN {X 0,Y 502.119,Z 1012.773,A -85,B 0,C 180,E1 -5846.796,E2 -5846.796} C_VEL
LIN {X 0,Y 502.064,Z 1014.171,A -85,B 0,C 180,E1 -5847.599,E2 -5847.599} C_VEL
LIN {X 0,Y 502.035,Z 1015.167,A -85,B 0,C 180,E1 -5848.401,E2 -5848.401} C_VEL
LIN {X 0,Y 501.98,Z 1015.984,A -85,B 0,C 180,E1 -5850.005,E2 -5850.005} C_VEL
LIN {X 0,Y 502.036,Z 1015.154,A -85,B 0,C 180,E1 -5851.61,E2 -5851.61} C_VEL
LIN {X 0,Y 502.066,Z 1014.153,A -85,B 0,C 180,E1 -5852.412,E2 -5852.412} C_VEL
LIN {X 0,Y 502.122,Z 1012.747,A -85,B 0,C 180,E1 -5853.215,E2 -5853.215} C_VEL
LIN {X 0,Y 502.127,Z 1009.775,A -85,B 0,C 180,E1 -5854.42,E2 -5854.42} C_VEL
LIN {X 0,Y 502.263,Z 1005.733,A -85,B 0,C 180,E1 -5855.626,E2 -5855.626} C_VEL
LIN {X 0,Y 502.34,Z 999.559,A -85,B 0,C 180,E1 -5857.016,E2 -5857.016} C_VEL
LIN {X 0,Y 502.519,Z 992.622,A -85,B 0,C 180,E1 -5858.247,E2 -5858.247} C_VEL
LIN {X 0,Y 502.795,Z 984.165,A -85,B 0,C 180,E1 -5859.458,E2 -5859.458} C_VEL
LIN {X 0,Y 503.063,Z 975.502,A -85,B 0,C 180,E1 -5860.469,E2 -5860.469} C_VEL
LIN {X 0,Y 503.442,Z 964.835,A -85,B 0,C 180,E1 -5861.479,E2 -5861.479} C_VEL
LIN {X 0,Y 503.797,Z 953.154,A -85,B 0,C 180,E1 -5862.368,E2 -5862.368} C_VEL
LIN {X 0,Y 504.057,Z 940.802,A -85,B 0,C 180,E1 -5863.1,E2 -5863.1} C_VEL
LIN {X 0,Y 504.392,Z 928.324,A -85,B 0,C 180,E1 -5863.655,E2 -5863.655} C_VEL
LIN {X 0,Y 504.692,Z 915.519,A -85,B 0,C 180,E1 -5864.058,E2 -5864.058} C_VEL
LIN {X 0,Y 504.889,Z 900.288,A -85,B 0,C 180,E1 -5864.335,E2 -5864.335} C_VEL
LIN {X 0,Y 505.313,Z 813.244,A -85,B 0,C 180,E1 -5865.572,E2 -5865.572} C_VEL
LIN {X 0,Y 503.72,Z 799.464,A -85,B 0,C 180,E1 -5865.83,E2 -5865.83} C_VEL
LIN {X 0,Y 504.302,Z 773.688,A -85,B 0,C 180,E1 -5868.91,E2 -5868.91} C_VEL
LIN {X 0,Y 504.959,Z 749.26,A -85,B 0,C 180,E1 -5871.862,E2 -5871.862} C_VEL
LIN {X 0,Y 505.508,Z 729.946,A -85,B 0,C 180,E1 -5874.217,E2 -5874.217} C_VEL
LIN {X 0,Y 506.262,Z 705.247,A -85,B 0,C 180,E1 -5877.269,E2 -5877.269} C_VEL
LIN {X 0,Y 502.778,Z 689.86,A -85,B 0,C 180,E1 -5879.42,E2 -5879.42} C_VEL
LIN {X 0,Y 502.758,Z 689.855,A -85,B 0,C 180,E1 -5882.09,E2 -5882.09} C_VEL
LIN {X 0,Y 502.717,Z 689.864,A -85,B 0,C 180,E1 -5884.976,E2 -5884.976} C_VEL
LIN {X 0,Y 502.756,Z 689.857,A -85,B 0,C 180,E1 -5888.48,E2 -5888.48} C_VEL
LIN {X 0,Y 502.764,Z 689.86,A -85,B 0,C 180,E1 -5891.075,E2 -5891.075} C_VEL
LIN {X 0,Y 502.792,Z 689.851,A -85,B 0,C 180,E1 -5894.531,E2 -5894.531} C_VEL
LIN {X 0,Y 502.781,Z 689.853,A -85,B 0,C 180,E1 -5897.859,E2 -5897.859} C_VEL
LIN {X 0,Y 502.796,Z 689.855,A -85,B 0,C 180,E1 -5901.023,E2 -5901.023} C_VEL
LIN {X 0,Y 502.778,Z 689.852,A -85,B 0,C 180,E1 -5904.172,E2 -5904.172} C_VEL
LIN {X 0,Y 502.845,Z 689.848,A -85,B 0,C 180,E1 -5906.995,E2 -5906.995} C_VEL
LIN {X 0,Y 502.828,Z 689.848,A -85,B 0,C 180,E1 -5910.066,E2 -5910.066} C_VEL
LIN {X 0,Y 502.812,Z 689.856,A -85,B 0,C 180,E1 -5913.455,E2 -5913.455} C_VEL
LIN {X 0,Y 502.783,Z 689.853,A -85,B 0,C 180,E1 -5916.086,E2 -5916.086} C_VEL
LIN {X 0,Y 502.795,Z 689.853,A -85,B 0,C 180,E1 -5918.689,E2 -5918.689} C_VEL
LIN {X 0,Y 502.837,Z 689.853,A -85,B 0,C 180,E1 -5921.248,E2 -5921.248} C_VEL
LIN {X 0,Y 502.869,Z 689.846,A -85,B 0,C 180,E1 -5924.656,E2 -5924.656} C_VEL
LIN {X 0,Y 502.878,Z 689.845,A -85,B 0,C 180,E1 -5924.759,E2 -5924.759} C_VEL
LIN {X 0,Y 505.178,Z 697.465,A -85,B 0,C 180,E1 -5924.961,E2 -5924.961} C_VEL
LIN {X 0,Y 504.686,Z 769.621,A -85,B 0,C 180,E1 -5926.075,E2 -5926.075} C_VEL
LIN {X 0,Y 504.651,Z 780.355,A -85,B 0,C 180,E1 -5926.357,E2 -5926.357} C_VEL
LIN {X 0,Y 504.508,Z 791.251,A -85,B 0,C 180,E1 -5926.763,E2 -5926.763} C_VEL
LIN {X 0,Y 504.332,Z 800.733,A -85,B 0,C 180,E1 -5927.222,E2 -5927.222} C_VEL
LIN {X 0,Y 504.129,Z 810.698,A -85,B 0,C 180,E1 -5927.832,E2 -5927.832} C_VEL
LIN {X 0,Y 503.873,Z 820.032,A -85,B 0,C 180,E1 -5928.536,E2 -5928.536} C_VEL
LIN {X 0,Y 503.687,Z 826.912,A -85,B 0,C 180,E1 -5929.142,E2 -5929.142} C_VEL
LIN {X 0,Y 503.364,Z 836.275,A -85,B 0,C 180,E1 -5930.152,E2 -5930.152} C_VEL
LIN {X 0,Y 503.224,Z 842.594,A -85,B 0,C 180,E1 -5930.96,E2 -5930.96} C_VEL
LIN {X 0,Y 503.02,Z 849.192,A -85,B 0,C 180,E1 -5931.969,E2 -5931.969} C_VEL
LIN {X 0,Y 502.837,Z 854.413,A -85,B 0,C 180,E1 -5932.917,E2 -5932.917} C_VEL
LIN {X 0,Y 502.782,Z 859.208,A -85,B 0,C 180,E1 -5933.982,E2 -5933.982} C_VEL
LIN {X 0,Y 502.534,Z 863.532,A -85,B 0,C 180,E1 -5935.187,E2 -5935.187} C_VEL
LIN {X 0,Y 502.446,Z 867.52,A -85,B 0,C 180,E1 -5936.793,E2 -5936.793} C_VEL
LIN {X 0,Y 502.442,Z 868.997,A -85,B 0,C 180,E1 -5937.595,E2 -5937.595} C_VEL
LIN {X 0,Y 502.388,Z 870.54,A -85,B 0,C 180,E1 -5939.198,E2 -5939.198} C_VEL
LIN {X 0,Y 502.355,Z 870.745,A -85,B 0,C 180,E1 -5940,E2 -5940} C_VEL
LIN {X 0,Y 502.317,Z 870.532,A -85,B 0,C 180,E1 -5940.802,E2 -5940.802} C_VEL
LIN {X 0,Y 502.332,Z 868.906,A -85,B 0,C 180,E1 -5942.406,E2 -5942.406} C_VEL
LIN {X 0,Y 502.48,Z 865.619,A -85,B 0,C 180,E1 -5944.01,E2 -5944.01} C_VEL
LIN {X 0,Y 502.528,Z 862.022,A -85,B 0,C 180,E1 -5945.216,E2 -5945.216} C_VEL
LIN {X 0,Y 502.712,Z 857.291,A -85,B 0,C 180,E1 -5946.422,E2 -5946.422} C_VEL
LIN {X 0,Y 502.796,Z 852.456,A -85,B 0,C 180,E1 -5947.429,E2 -5947.429} C_VEL
LIN {X 0,Y 503.016,Z 846.594,A -85,B 0,C 180,E1 -5948.436,E2 -5948.436} C_VEL
LIN {X 0,Y 503.218,Z 839.506,A -85,B 0,C 180,E1 -5949.445,E2 -5949.445} C_VEL
LIN {X 0,Y 503.446,Z 830.889,A -85,B 0,C 180,E1 -5950.456,E2 -5950.456} C_VEL
LIN {X 0,Y 503.723,Z 822.61,A -85,B 0,C 180,E1 -5951.264,E2 -5951.264} C_VEL
LIN {X 0,Y 503.933,Z 813.959,A -85,B 0,C 180,E1 -5951.973,E2 -5951.973} C_VEL
LIN {X 0,Y 504.203,Z 803.912,A -85,B 0,C 180,E1 -5952.646,E2 -5952.646} C_VEL
LIN {X 0,Y 504.42,Z 793.8,A -85,B 0,C 180,E1 -5953.188,E2 -5953.188} C_VEL
LIN {X 0,Y 504.585,Z 783.506,A -85,B 0,C 180,E1 -5953.62,E2 -5953.62} C_VEL
LIN {X 0,Y 504.679,Z 772.798,A -85,B 0,C 180,E1 -5953.951,E2 -5953.951} C_VEL
LIN {X 0,Y 504.802,Z 760.192,A -85,B 0,C 180,E1 -5954.204,E2 -5954.204} C_VEL
LIN {X 0,Y 505.047,Z 696.495,A -85,B 0,C 180,E1 -5955.157,E2 -5955.157} C_VEL
LIN {X 0,Y 502.859,Z 689.846,A -85,B 0,C 180,E1 -5955.34,E2 -5955.34} C_VEL
LIN {X 0,Y 502.84,Z 689.847,A -85,B 0,C 180,E1 -5958.115,E2 -5958.115} C_VEL
LIN {X 0,Y 502.843,Z 689.85,A -85,B 0,C 180,E1 -5960.536,E2 -5960.536} C_VEL
LIN {X 0,Y 502.8,Z 689.854,A -85,B 0,C 180,E1 -5963.04,E2 -5963.04} C_VEL
LIN {X 0,Y 502.803,Z 689.849,A -85,B 0,C 180,E1 -5965.678,E2 -5965.678} C_VEL
LIN {X 0,Y 502.809,Z 689.849,A -85,B 0,C 180,E1 -5968.375,E2 -5968.375} C_VEL
LIN {X 0,Y 502.809,Z 689.853,A -85,B 0,C 180,E1 -5971.143,E2 -5971.143} C_VEL
LIN {X 0,Y 502.8,Z 689.848,A -85,B 0,C 180,E1 -5973.994,E2 -5973.994} C_VEL
LIN {X 0,Y 502.779,Z 689.857,A -85,B 0,C 180,E1 -5977.174,E2 -5977.174} C_VEL
LIN {X 0,Y 502.786,Z 689.85,A -85,B 0,C 180,E1 -5980.016,E2 -5980.016} C_VEL
LIN {X 0,Y 502.766,Z 689.857,A -85,B 0,C 180,E1 -5983.232,E2 -5983.232} C_VEL
LIN {X 0,Y 502.782,Z 689.851,A -85,B 0,C 180,E1 -5985.657,E2 -5985.657} C_VEL
LIN {X 0,Y 502.749,Z 689.854,A -85,B 0,C 180,E1 -5986.327,E2 -5986.327} C_VEL
LIN {X 0,Y 502.086,Z 689.944,A -85,B 0,C 180,E1 -5986.996,E2 -5986.996} C_VEL
LIN {X 0,Y 499.229,Z 690.298,A -85,B 0,C 180,E1 -5988.082,E2 -5988.082} C_VEL
LIN {X 0,Y 496.828,Z 690.598,A -85,B 0,C 180,E1 -5988.958,E2 -5988.958} C_VEL
LIN {X 0,Y 495.82,Z 690.719,A -85,B 0,C 180,E1 -5989.634,E2 -5989.634} C_VEL
LIN {X 0,Y 495.751,Z 690.726,A -85,B 0,C 180,E1 -5989.863,E2 -5989.863} C_VEL
LIN {X 0,Y 495.71,Z 690.732,A -85,B 0,C 180,E1 -5992.556,E2 -5992.556} C_VEL
LIN {X 0,Y 495.767,Z 690.728,A -85,B 0,C 180,E1 -5995.452,E2 -5995.452} C_VEL
LIN {X 0,Y 495.744,Z 690.727,A -85,B 0,C 180,E1 -5998.359,E2 -5998.359} C_VEL
LIN {X 0,Y 495.732,Z 690.733,A -85,B 0,C 180,E1 -6001.519,E2 -6001.519} C_VEL
LIN {X 0,Y 495.723,Z 690.734,A -85,B 0,C 180,E1 -6004.825,E2 -6004.825} C_VEL
LIN {X 0,Y 495.745,Z 690.736,A -85,B 0,C 180,E1 -6007.491,E2 -6007.491} C_VEL
LIN {X 0,Y 495.716,Z 690.734,A -85,B 0,C 180,E1 -6010.103,E2 -6010.103} C_VEL
LIN {X 0,Y 495.732,Z 690.733,A -85,B 0,C 180,E1 -6012.675,E2 -6012.675} C_VEL
LIN {X 0,Y 495.768,Z 690.729,A -85,B 0,C 180,E1 -6014.385,E2 -6014.385} C_VEL
LIN {X 0,Y 498.707,Z 699.988,A -85,B 0,C 180,E1 -6014.625,E2 -6014.625} C_VEL
LIN {X 0,Y 498.198,Z 771.498,A -85,B 0,C 180,E1 -6015.677,E2 -6015.677} C_VEL
LIN {X 0,Y 498.241,Z 784.637,A -85,B 0,C 180,E1 -6016.043,E2 -6016.043} C_VEL
LIN {X 0,Y 498.069,Z 796.68,A -85,B 0,C 180,E1 -6016.533,E2 -6016.533} C_VEL
LIN {X 0,Y 497.851,Z 808.285,A -85,B 0,C 180,E1 -6017.168,E2 -6017.168} C_VEL
LIN {X 0,Y 497.487,Z 819.564,A -85,B 0,C 180,E1 -6017.968,E2 -6017.968} C_VEL
LIN {X 0,Y 497.169,Z 829.914,A -85,B 0,C 180,E1 -6018.891,E2 -6018.891} C_VEL
LIN {X 0,Y 496.873,Z 838.356,A -85,B 0,C 180,E1 -6019.812,E2 -6019.812} C_VEL
LIN {X 0,Y 496.551,Z 846.123,A -85,B 0,C 180,E1 -6020.833,E2 -6020.833} C_VEL
LIN {X 0,Y 496.207,Z 853.821,A -85,B 0,C 180,E1 -6022.078,E2 -6022.078} C_VEL
LIN {X 0,Y 496.102,Z 859.479,A -85,B 0,C 180,E1 -6023.22,E2 -6023.22} C_VEL
LIN {X 0,Y 495.823,Z 865.258,A -85,B 0,C 180,E1 -6024.709,E2 -6024.709} C_VEL
LIN {X 0,Y 495.646,Z 868.795,A -85,B 0,C 180,E1 -6025.929,E2 -6025.929} C_VEL
LIN {X 0,Y 495.565,Z 870.622,A -85,B 0,C 180,E1 -6026.743,E2 -6026.743} C_VEL
LIN {X 0,Y 495.558,Z 871.996,A -85,B 0,C 180,E1 -6027.556,E2 -6027.556} C_VEL
LIN {X 0,Y 495.522,Z 873.578,A -85,B 0,C 180,E1 -6029.182,E2 -6029.182} C_VEL
LIN {X 0,Y 495.506,Z 873.814,A -85,B 0,C 180,E1 -6029.995,E2 -6029.995} C_VEL
LIN {X 0,Y 495.589,Z 873.064,A -85,B 0,C 180,E1 -6031.62,E2 -6031.62} C_VEL
LIN {X 0,Y 495.558,Z 870.822,A -85,B 0,C 180,E1 -6033.246,E2 -6033.246} C_VEL
LIN {X 0,Y 495.697,Z 868.019,A -85,B 0,C 180,E1 -6034.467,E2 -6034.467} C_VEL
LIN {X 0,Y 495.875,Z 864.216,A -85,B 0,C 180,E1 -6035.688,E2 -6035.688} C_VEL
LIN {X 0,Y 496.059,Z 858.751,A -85,B 0,C 180,E1 -6037.036,E2 -6037.036} C_VEL
LIN {X 0,Y 496.312,Z 851.941,A -85,B 0,C 180,E1 -6038.34,E2 -6038.34} C_VEL
LIN {X 0,Y 496.659,Z 843.933,A -85,B 0,C 180,E1 -6039.565,E2 -6039.565} C_VEL
LIN {X 0,Y 496.967,Z 835.728,A -85,B 0,C 180,E1 -6040.587,E2 -6040.587} C_VEL
LIN {X 0,Y 497.298,Z 825.578,A -85,B 0,C 180,E1 -6041.612,E2 -6041.612} C_VEL
LIN {X 0,Y 497.717,Z 815.134,A -85,B 0,C 180,E1 -6042.456,E2 -6042.456} C_VEL
LIN {X 0,Y 497.958,Z 803.9,A -85,B 0,C 180,E1 -6043.182,E2 -6043.182} C_VEL
LIN {X 0,Y 498.128,Z 792.062,A -85,B 0,C 180,E1 -6043.767,E2 -6043.767} C_VEL
LIN {X 0,Y 498.289,Z 778.73,A -85,B 0,C 180,E1 -6044.231,E2 -6044.231} C_VEL
LIN {X 0,Y 498.319,Z 765.52,A -85,B 0,C 180,E1 -6044.517,E2 -6044.517} C_VEL
LIN {X 0,Y 498.634,Z 699.079,A -85,B 0,C 180,E1 -6045.482,E2 -6045.482} C_VEL
LIN {X 0,Y 495.777,Z 690.729,A -85,B 0,C 180,E1 -6045.723,E2 -6045.723} C_VEL
LIN {X 0,Y 495.766,Z 690.734,A -85,B 0,C 180,E1 -6049.022,E2 -6049.022} C_VEL
LIN {X 0,Y 495.723,Z 690.731,A -85,B 0,C 180,E1 -6051.622,E2 -6051.622} C_VEL
LIN {X 0,Y 495.694,Z 690.734,A -85,B 0,C 180,E1 -6054.27,E2 -6054.27} C_VEL
LIN {X 0,Y 495.758,Z 690.731,A -85,B 0,C 180,E1 -6056.969,E2 -6056.969} C_VEL
LIN {X 0,Y 495.736,Z 690.73,A -85,B 0,C 180,E1 -6059.74,E2 -6059.74} C_VEL
LIN {X 0,Y 495.735,Z 690.73,A -85,B 0,C 180,E1 -6062.588,E2 -6062.588} C_VEL
LIN {X 0,Y 495.719,Z 690.738,A -85,B 0,C 180,E1 -6065.531,E2 -6065.531} C_VEL
LIN {X 0,Y 495.727,Z 690.723,A -85,B 0,C 180,E1 -6068.763,E2 -6068.763} C_VEL
LIN {X 0,Y 495.741,Z 690.736,A -85,B 0,C 180,E1 -6071.772,E2 -6071.772} C_VEL
LIN {X 0,Y 495.701,Z 690.729,A -85,B 0,C 180,E1 -6075.133,E2 -6075.133} C_VEL
LIN {X 0,Y 495.734,Z 690.733,A -85,B 0,C 180,E1 -6078.216,E2 -6078.216} C_VEL
LIN {X 0,Y 495.729,Z 690.73,A -85,B 0,C 180,E1 -6081.223,E2 -6081.223} C_VEL
LIN {X 0,Y 495.699,Z 690.734,A -85,B 0,C 180,E1 -6084.458,E2 -6084.458} C_VEL
LIN {X 0,Y 495.709,Z 690.732,A -85,B 0,C 180,E1 -6087.401,E2 -6087.401} C_VEL
LIN {X 0,Y 495.718,Z 690.734,A -85,B 0,C 180,E1 -6090.25,E2 -6090.25} C_VEL
LIN {X 0,Y 495.767,Z 690.725,A -85,B 0,C 180,E1 -6093.244,E2 -6093.244} C_VEL
LIN {X 0,Y 495.689,Z 690.735,A -85,B 0,C 180,E1 -6095.722,E2 -6095.722} C_VEL
LIN {X 0,Y 495.683,Z 690.743,A -85,B 0,C 180,E1 -6098.368,E2 -6098.368} C_VEL
LIN {X 0,Y 495.712,Z 690.731,A -85,B 0,C 180,E1 -6100.969,E2 -6100.969} C_VEL
LIN {X 0,Y 495.712,Z 690.729,A -85,B 0,C 180,E1 -6103.528,E2 -6103.528} C_VEL
LIN {X 0,Y 495.738,Z 690.731,A -85,B 0,C 180,E1 -6106.054,E2 -6106.054} C_VEL
LIN {X 0,Y 495.805,Z 690.726,A -85,B 0,C 180,E1 -6108.554,E2 -6108.554} C_VEL
LIN {X 0,Y 495.803,Z 690.721,A -85,B 0,C 180,E1 -6111.851,E2 -6111.851} C_VEL
LIN {X 0,Y 495.843,Z 690.718,A -85,B 0,C 180,E1 -6114.306,E2 -6114.306} C_VEL
LIN {X 0,Y 495.921,Z 690.707,A -85,B 0,C 180,E1 -6117.563,E2 -6117.563} C_VEL
LIN {X 0,Y 495.916,Z 690.708,A -85,B 0,C 180,E1 -6120,E2 -6120} C_VEL
LIN {X 0,Y 495.921,Z 690.705,A -85,B 0,C 180,E1 -6122.437,E2 -6122.437} C_VEL
LIN {X 0,Y 495.843,Z 690.719,A -85,B 0,C 180,E1 -6125.694,E2 -6125.694} C_VEL
LIN {X 0,Y 495.802,Z 690.719,A -85,B 0,C 180,E1 -6128.149,E2 -6128.149} C_VEL
LIN {X 0,Y 495.804,Z 690.729,A -85,B 0,C 180,E1 -6131.446,E2 -6131.446} C_VEL
LIN {X 0,Y 495.731,Z 690.73,A -85,B 0,C 180,E1 -6134.785,E2 -6134.785} C_VEL
LIN {X 0,Y 495.717,Z 690.737,A -85,B 0,C 180,E1 -6137.321,E2 -6137.321} C_VEL
LIN {X 0,Y 495.706,Z 690.733,A -85,B 0,C 180,E1 -6139.893,E2 -6139.893} C_VEL
LIN {X 0,Y 495.696,Z 690.733,A -85,B 0,C 180,E1 -6142.866,E2 -6142.866} C_VEL
LIN {X 0,Y 495.739,Z 690.731,A -85,B 0,C 180,E1 -6146.071,E2 -6146.071} C_VEL
LIN {X 0,Y 495.715,Z 690.731,A -85,B 0,C 180,E1 -6148.819,E2 -6148.819} C_VEL
LIN {X 0,Y 495.701,Z 690.737,A -85,B 0,C 180,E1 -6151.732,E2 -6151.732} C_VEL
LIN {X 0,Y 495.716,Z 690.732,A -85,B 0,C 180,E1 -6154.7,E2 -6154.7} C_VEL
LIN {X 0,Y 495.677,Z 690.737,A -85,B 0,C 180,E1 -6157.566,E2 -6157.566} C_VEL
LIN {X 0,Y 495.752,Z 690.729,A -85,B 0,C 180,E1 -6160.059,E2 -6160.059} C_VEL
LIN {X 0,Y 495.713,Z 690.734,A -85,B 0,C 180,E1 -6162.885,E2 -6162.885} C_VEL
LIN {X 0,Y 495.689,Z 690.739,A -85,B 0,C 180,E1 -6166.005,E2 -6166.005} C_VEL
LIN {X 0,Y 495.728,Z 690.737,A -85,B 0,C 180,E1 -6168.711,E2 -6168.711} C_VEL
LIN {X 0,Y 495.713,Z 690.733,A -85,B 0,C 180,E1 -6171.415,E2 -6171.415} C_VEL
LIN {X 0,Y 495.718,Z 690.739,A -85,B 0,C 180,E1 -6174.469,E2 -6174.469} C_VEL
LIN {X 0,Y 495.734,Z 690.734,A -85,B 0,C 180,E1 -6177.412,E2 -6177.412} C_VEL
LIN {X 0,Y 495.782,Z 690.835,A -85,B 0,C 180,E1 -6180.395,E2 -6180.395} C_VEL
LIN {X 0,Y 499.298,Z 706.909,A -85,B 0,C 180,E1 -6182.651,E2 -6182.651} C_VEL
LIN {X 0,Y 498.75,Z 725.593,A -85,B 0,C 180,E1 -6185,E2 -6185} C_VEL
LIN {X 0,Y 498.007,Z 748.427,A -85,B 0,C 180,E1 -6187.828,E2 -6187.828} C_VEL
LIN {X 0,Y 497.321,Z 772.838,A -85,B 0,C 180,E1 -6190.826,E2 -6190.826} C_VEL
LIN {X 0,Y 496.699,Z 795.365,A -85,B 0,C 180,E1 -6193.568,E2 -6193.568} C_VEL
LIN {X 0,Y 496.679,Z 798.808,A -85,B 0,C 180,E1 -6193.958,E2 -6193.958} C_VEL
LIN {X 0,Y 498.49,Z 814.807,A -85,B 0,C 180,E1 -6194.247,E2 -6194.247} C_VEL
LIN {X 0,Y 497.921,Z 909.349,A -85,B 0,C 180,E1 -6195.628,E2 -6195.628} C_VEL
LIN {X 0,Y 497.608,Z 922.603,A -85,B 0,C 180,E1 -6195.984,E2 -6195.984} C_VEL
LIN {X 0,Y 497.236,Z 935.953,A -85,B 0,C 180,E1 -6196.52,E2 -6196.52} C_VEL
LIN {X 0,Y 496.884,Z 948.289,A -85,B 0,C 180,E1 -6197.204,E2 -6197.204} C_VEL
LIN {X 0,Y 496.55,Z 960.271,A -85,B 0,C 180,E1 -6198.06,E2 -6198.06} C_VEL
LIN {X 0,Y 496.171,Z 970.612,A -85,B 0,C 180,E1 -6198.982,E2 -6198.982} C_VEL
LIN {X 0,Y 495.852,Z 979.946,A -85,B 0,C 180,E1 -6200.007,E2 -6200.007} C_VEL
LIN {X 0,Y 495.543,Z 989.057,A -85,B 0,C 180,E1 -6201.236,E2 -6201.236} C_VEL
LIN {X 0,Y 495.311,Z 996.408,A -85,B 0,C 180,E1 -6202.464,E2 -6202.464} C_VEL
LIN {X 0,Y 495.198,Z 1002.398,A -85,B 0,C 180,E1 -6203.718,E2 -6203.718} C_VEL
LIN {X 0,Y 495.148,Z 1006.224,A -85,B 0,C 180,E1 -6204.712,E2 -6204.712} C_VEL
LIN {X 0,Y 495.087,Z 1009.929,A -85,B 0,C 180,E1 -6205.936,E2 -6205.936} C_VEL
LIN {X 0,Y 495.073,Z 1011.842,A -85,B 0,C 180,E1 -6206.75,E2 -6206.75} C_VEL
LIN {X 0,Y 495.014,Z 1013.268,A -85,B 0,C 180,E1 -6207.564,E2 -6207.564} C_VEL
LIN {X 0,Y 494.985,Z 1014.287,A -85,B 0,C 180,E1 -6208.378,E2 -6208.378} C_VEL
LIN {X 0,Y 494.943,Z 1014.903,A -85,B 0,C 180,E1 -6209.192,E2 -6209.192} C_VEL
LIN {X 0,Y 494.933,Z 1015.121,A -85,B 0,C 180,E1 -6210.005,E2 -6210.005} C_VEL
LIN {X 0,Y 494.943,Z 1014.896,A -85,B 0,C 180,E1 -6210.819,E2 -6210.819} C_VEL
LIN {X 0,Y 494.986,Z 1014.274,A -85,B 0,C 180,E1 -6211.633,E2 -6211.633} C_VEL
LIN {X 0,Y 495.016,Z 1013.25,A -85,B 0,C 180,E1 -6212.446,E2 -6212.446} C_VEL
LIN {X 0,Y 495.076,Z 1011.817,A -85,B 0,C 180,E1 -6213.26,E2 -6213.26} C_VEL
LIN {X 0,Y 495.072,Z 1008.794,A -85,B 0,C 180,E1 -6214.483,E2 -6214.483} C_VEL
LIN {X 0,Y 495.2,Z 1004.722,A -85,B 0,C 180,E1 -6215.707,E2 -6215.707} C_VEL
LIN {X 0,Y 495.277,Z 998.544,A -85,B 0,C 180,E1 -6217.117,E2 -6217.117} C_VEL
LIN {X 0,Y 495.464,Z 991.605,A -85,B 0,C 180,E1 -6218.365,E2 -6218.365} C_VEL
LIN {X 0,Y 495.721,Z 983.142,A -85,B 0,C 180,E1 -6219.594,E2 -6219.594} C_VEL
LIN {X 0,Y 496.015,Z 974.48,A -85,B 0,C 180,E1 -6220.619,E2 -6220.619} C_VEL
LIN {X 0,Y 496.406,Z 963.81,A -85,B 0,C 180,E1 -6221.644,E2 -6221.644} C_VEL
LIN {X 0,Y 496.794,Z 952.136,A -85,B 0,C 180,E1 -6222.545,E2 -6222.545} C_VEL
LIN {X 0,Y 497.087,Z 939.781,A -85,B 0,C 180,E1 -6223.287,E2 -6223.287} C_VEL
LIN {X 0,Y 497.475,Z 927.309,A -85,B 0,C 180,E1 -6223.849,E2 -6223.849} C_VEL
LIN {X 0,Y 497.804,Z 914.505,A -85,B 0,C 180,E1 -6224.256,E2 -6224.256} C_VEL
LIN {X 0,Y 497.992,Z 901.069,A -85,B 0,C 180,E1 -6224.512,E2 -6224.512} C_VEL
LIN {X 0,Y 498.418,Z 813.087,A -85,B 0,C 180,E1 -6225.78,E2 -6225.78} C_VEL
LIN {X 0,Y 496.667,Z 798.449,A -85,B 0,C 180,E1 -6226.057,E2 -6226.057} C_VEL
LIN {X 0,Y 497.285,Z 774.496,A -85,B 0,C 180,E1 -6228.973,E2 -6228.973} C_VEL
LIN {X 0,Y 497.99,Z 750.095,A -85,B 0,C 180,E1 -6231.966,E2 -6231.966} C_VEL
LIN {X 0,Y 498.58,Z 730.787,A -85,B 0,C 180,E1 -6234.354,E2 -6234.354} C_VEL
LIN {X 0,Y 499.354,Z 706.898,A -85,B 0,C 180,E1 -6237.348,E2 -6237.348} C_VEL
LIN {X 0,Y 495.727,Z 690.737,A -85,B 0,C 180,E1 -6239.636,E2 -6239.636} C_VEL
LIN {X 0,Y 495.723,Z 690.731,A -85,B 0,C 180,E1 -6242.601,E2 -6242.601} C_VEL
LIN {X 0,Y 495.667,Z 690.736,A -85,B 0,C 180,E1 -6245.548,E2 -6245.548} C_VEL
LIN {X 0,Y 495.734,Z 690.734,A -85,B 0,C 180,E1 -6248.764,E2 -6248.764} C_VEL
LIN {X 0,Y 495.714,Z 690.734,A -85,B 0,C 180,E1 -6251.789,E2 -6251.789} C_VEL
LIN {X 0,Y 495.746,Z 690.735,A -85,B 0,C 180,E1 -6255.143,E2 -6255.143} C_VEL
LIN {X 0,Y 495.738,Z 690.729,A -85,B 0,C 180,E1 -6258.217,E2 -6258.217} C_VEL
LIN {X 0,Y 495.753,Z 690.734,A -85,B 0,C 180,E1 -6261.237,E2 -6261.237} C_VEL
LIN {X 0,Y 495.752,Z 690.728,A -85,B 0,C 180,E1 -6264.462,E2 -6264.462} C_VEL
LIN {X 0,Y 495.78,Z 690.731,A -85,B 0,C 180,E1 -6267.406,E2 -6267.406} C_VEL
LIN {X 0,Y 495.776,Z 690.726,A -85,B 0,C 180,E1 -6270.254,E2 -6270.254} C_VEL
LIN {X 0,Y 495.772,Z 690.732,A -85,B 0,C 180,E1 -6273.267,E2 -6273.267} C_VEL
LIN {X 0,Y 495.753,Z 690.729,A -85,B 0,C 180,E1 -6276.613,E2 -6276.613} C_VEL
LIN {X 0,Y 495.793,Z 690.731,A -85,B 0,C 180,E1 -6279.325,E2 -6279.325} C_VEL
LIN {X 0,Y 495.793,Z 690.728,A -85,B 0,C 180,E1 -6281.829,E2 -6281.829} C_VEL
LIN {X 0,Y 495.826,Z 690.769,A -85,B 0,C 180,E1 -6284.554,E2 -6284.554} C_VEL
LIN {X 0,Y 498.242,Z 698.165,A -85,B 0,C 180,E1 -6284.754,E2 -6284.754} C_VEL
LIN {X 0,Y 497.778,Z 770.784,A -85,B 0,C 180,E1 -6285.904,E2 -6285.904} C_VEL
LIN {X 0,Y 497.726,Z 782.256,A -85,B 0,C 180,E1 -6286.215,E2 -6286.215} C_VEL
LIN {X 0,Y 497.599,Z 792.952,A -85,B 0,C 180,E1 -6286.628,E2 -6286.628} C_VEL
LIN {X 0,Y 497.434,Z 801.839,A -85,B 0,C 180,E1 -6287.066,E2 -6287.066} C_VEL
LIN {X 0,Y 497.232,Z 811.544,A -85,B 0,C 180,E1 -6287.666,E2 -6287.666} C_VEL
LIN {X 0,Y 496.966,Z 820.872,A -85,B 0,C 180,E1 -6288.374,E2 -6288.374} C_VEL
LIN {X 0,Y 496.703,Z 829.749,A -85,B 0,C 180,E1 -6289.194,E2 -6289.194} C_VEL
LIN {X 0,Y 496.457,Z 837.193,A -85,B 0,C 180,E1 -6290.014,E2 -6290.014} C_VEL
LIN {X 0,Y 496.181,Z 844.906,A -85,B 0,C 180,E1 -6291.036,E2 -6291.036} C_VEL
LIN {X 0,Y 495.989,Z 851.298,A -85,B 0,C 180,E1 -6292.059,E2 -6292.059} C_VEL
LIN {X 0,Y 495.865,Z 855.408,A -85,B 0,C 180,E1 -6292.816,E2 -6292.816} C_VEL
LIN {X 0,Y 495.802,Z 860.223,A -85,B 0,C 180,E1 -6293.897,E2 -6293.897} C_VEL
LIN {X 0,Y 495.534,Z 864.565,A -85,B 0,C 180,E1 -6295.118,E2 -6295.118} C_VEL
LIN {X 0,Y 495.435,Z 868.565,A -85,B 0,C 180,E1 -6296.747,E2 -6296.747} C_VEL
LIN {X 0,Y 495.439,Z 870.039,A -85,B 0,C 180,E1 -6297.561,E2 -6297.561} C_VEL
LIN {X 0,Y 495.385,Z 871.577,A -85,B 0,C 180,E1 -6299.187,E2 -6299.187} C_VEL
LIN {X 0,Y 495.351,Z 871.774,A -85,B 0,C 180,E1 -6300,E2 -6300} C_VEL
LIN {X 0,Y 495.321,Z 871.552,A -85,B 0,C 180,E1 -6300.813,E2 -6300.813} C_VEL
LIN {X 0,Y 495.309,Z 869.905,A -85,B 0,C 180,E1 -6302.44,E2 -6302.44} C_VEL
LIN {X 0,Y 495.464,Z 866.586,A -85,B 0,C 180,E1 -6304.067,E2 -6304.067} C_VEL
LIN {X 0,Y 495.528,Z 862.958,A -85,B 0,C 180,E1 -6305.29,E2 -6305.29} C_VEL
LIN {X 0,Y 495.73,Z 858.184,A -85,B 0,C 180,E1 -6306.512,E2 -6306.512} C_VEL
LIN {X 0,Y 495.825,Z 853.318,A -85,B 0,C 180,E1 -6307.534,E2 -6307.534} C_VEL
LIN {X 0,Y 496.057,Z 847.412,A -85,B 0,C 180,E1 -6308.555,E2 -6308.555} C_VEL
LIN {X 0,Y 496.269,Z 840.275,A -85,B 0,C 180,E1 -6309.579,E2 -6309.579} C_VEL
LIN {X 0,Y 496.514,Z 831.604,A -85,B 0,C 180,E1 -6310.604,E2 -6310.604} C_VEL
LIN {X 0,Y 496.81,Z 823.261,A -85,B 0,C 180,E1 -6311.423,E2 -6311.423} C_VEL
LIN {X 0,Y 497.033,Z 814.532,A -85,B 0,C 180,E1 -6312.142,E2 -6312.142} C_VEL
LIN {X 0,Y 497.298,Z 804.848,A -85,B 0,C 180,E1 -6312.797,E2 -6312.797} C_VEL
LIN {X 0,Y 497.523,Z 795.272,A -85,B 0,C 180,E1 -6313.322,E2 -6313.322} C_VEL
LIN {X 0,Y 497.691,Z 784.413,A -85,B 0,C 180,E1 -6313.786,E2 -6313.786} C_VEL
LIN {X 0,Y 497.788,Z 773.713,A -85,B 0,C 180,E1 -6314.122,E2 -6314.122} C_VEL
LIN {X 0,Y 497.916,Z 761.162,A -85,B 0,C 180,E1 -6314.379,E2 -6314.379} C_VEL
LIN {X 0,Y 498.363,Z 698.848,A -85,B 0,C 180,E1 -6315.327,E2 -6315.327} C_VEL
LIN {X 0,Y 495.828,Z 690.721,A -85,B 0,C 180,E1 -6315.554,E2 -6315.554} C_VEL
LIN {X 0,Y 495.791,Z 690.728,A -85,B 0,C 180,E1 -6319.028,E2 -6319.028} C_VEL
LIN {X 0,Y 495.753,Z 690.727,A -85,B 0,C 180,E1 -6321.629,E2 -6321.629} C_VEL
LIN {X 0,Y 495.731,Z 690.732,A -85,B 0,C 180,E1 -6324.276,E2 -6324.276} C_VEL
LIN {X 0,Y 495.763,Z 690.732,A -85,B 0,C 180,E1 -6326.977,E2 -6326.977} C_VEL
LIN {X 0,Y 495.778,Z 690.724,A -85,B 0,C 180,E1 -6330.146,E2 -6330.146} C_VEL
LIN {X 0,Y 495.766,Z 690.729,A -85,B 0,C 180,E1 -6333.236,E2 -6333.236} C_VEL
LIN {X 0,Y 495.726,Z 690.729,A -85,B 0,C 180,E1 -6336.086,E2 -6336.086} C_VEL
LIN {X 0,Y 495.772,Z 690.73,A -85,B 0,C 180,E1 -6338.766,E2 -6338.766} C_VEL
LIN {X 0,Y 495.741,Z 690.727,A -85,B 0,C 180,E1 -6341.783,E2 -6341.783} C_VEL
LIN {X 0,Y 495.749,Z 690.733,A -85,B 0,C 180,E1 -6345.14,E2 -6345.14} C_VEL
LIN {X 0,Y 495.739,Z 690.727,A -85,B 0,C 180,E1 -6348.213,E2 -6348.213} C_VEL
LIN {X 0,Y 495.751,Z 690.726,A -85,B 0,C 180,E1 -6349.863,E2 -6349.863} C_VEL
LIN {X 0,Y 495.107,Z 690.808,A -85,B 0,C 180,E1 -6350.541,E2 -6350.541} C_VEL
LIN {X 0,Y 492.221,Z 691.167,A -85,B 0,C 180,E1 -6351.642,E2 -6351.642} C_VEL
LIN {X 0,Y 489.77,Z 691.472,A -85,B 0,C 180,E1 -6352.529,E2 -6352.529} C_VEL
LIN {X 0,Y 488.729,Z 691.607,A -85,B 0,C 180,E1 -6353.214,E2 -6353.214} C_VEL
LIN {X 0,Y 488.651,Z 691.611,A -85,B 0,C 180,E1 -6353.447,E2 -6353.447} C_VEL
LIN {X 0,Y 488.719,Z 691.602,A -85,B 0,C 180,E1 -6355.882,E2 -6355.882} C_VEL
LIN {X 0,Y 488.673,Z 691.611,A -85,B 0,C 180,E1 -6358.815,E2 -6358.815} C_VEL
LIN {X 0,Y 488.689,Z 691.609,A -85,B 0,C 180,E1 -6361.664,E2 -6361.664} C_VEL
LIN {X 0,Y 488.702,Z 691.61,A -85,B 0,C 180,E1 -6364.959,E2 -6364.959} C_VEL
LIN {X 0,Y 488.694,Z 691.608,A -85,B 0,C 180,E1 -6368.039,E2 -6368.039} C_VEL
LIN {X 0,Y 488.68,Z 691.611,A -85,B 0,C 180,E1 -6370.68,E2 -6370.68} C_VEL
LIN {X 0,Y 488.695,Z 691.615,A -85,B 0,C 180,E1 -6373.28,E2 -6373.28} C_VEL
LIN {X 0,Y 488.7,Z 691.61,A -85,B 0,C 180,E1 -6374.138,E2 -6374.138} C_VEL
LIN {X 0,Y 491.882,Z 701.378,A -85,B 0,C 180,E1 -6374.411,E2 -6374.411} C_VEL
LIN {X 0,Y 491.363,Z 772.525,A -85,B 0,C 180,E1 -6375.473,E2 -6375.473} C_VEL
LIN {X 0,Y 491.419,Z 785.654,A -85,B 0,C 180,E1 -6375.845,E2 -6375.845} C_VEL
LIN {X 0,Y 491.245,Z 797.691,A -85,B 0,C 180,E1 -6376.342,E2 -6376.342} C_VEL
LIN {X 0,Y 491.001,Z 809.289,A -85,B 0,C 180,E1 -6376.986,E2 -6376.986} C_VEL
LIN {X 0,Y 490.619,Z 820.572,A -85,B 0,C 180,E1 -6377.797,E2 -6377.797} C_VEL
LIN {X 0,Y 490.278,Z 830.921,A -85,B 0,C 180,E1 -6378.732,E2 -6378.732} C_VEL
LIN {X 0,Y 489.964,Z 839.361,A -85,B 0,C 180,E1 -6379.666,E2 -6379.666} C_VEL
LIN {X 0,Y 489.618,Z 847.128,A -85,B 0,C 180,E1 -6380.702,E2 -6380.702} C_VEL
LIN {X 0,Y 489.247,Z 854.826,A -85,B 0,C 180,E1 -6381.965,E2 -6381.965} C_VEL
LIN {X 0,Y 489.128,Z 860.481,A -85,B 0,C 180,E1 -6383.122,E2 -6383.122} C_VEL
LIN {X 0,Y 488.837,Z 866.261,A -85,B 0,C 180,E1 -6384.633,E2 -6384.633} C_VEL
LIN {X 0,Y 488.635,Z 869.799,A -85,B 0,C 180,E1 -6385.871,E2 -6385.871} C_VEL
LIN {X 0,Y 488.548,Z 871.626,A -85,B 0,C 180,E1 -6386.696,E2 -6386.696} C_VEL
LIN {X 0,Y 488.544,Z 872.999,A -85,B 0,C 180,E1 -6387.521,E2 -6387.521} C_VEL
LIN {X 0,Y 488.504,Z 874.58,A -85,B 0,C 180,E1 -6389.17,E2 -6389.17} C_VEL
LIN {X 0,Y 488.488,Z 874.815,A -85,B 0,C 180,E1 -6389.995,E2 -6389.995} C_VEL
LIN {X 0,Y 488.578,Z 874.064,A -85,B 0,C 180,E1 -6391.643,E2 -6391.643} C_VEL
LIN {X 0,Y 488.54,Z 871.823,A -85,B 0,C 180,E1 -6393.293,E2 -6393.293} C_VEL
LIN {X 0,Y 488.691,Z 869.02,A -85,B 0,C 180,E1 -6394.531,E2 -6394.531} C_VEL
LIN {X 0,Y 488.892,Z 865.216,A -85,B 0,C 180,E1 -6395.769,E2 -6395.769} C_VEL
LIN {X 0,Y 489.086,Z 859.747,A -85,B 0,C 180,E1 -6397.137,E2 -6397.137} C_VEL
LIN {X 0,Y 489.361,Z 852.941,A -85,B 0,C 180,E1 -6398.459,E2 -6398.459} C_VEL
LIN {X 0,Y 489.736,Z 844.932,A -85,B 0,C 180,E1 -6399.701,E2 -6399.701} C_VEL
LIN {X 0,Y 490.064,Z 836.726,A -85,B 0,C 180,E1 -6400.738,E2 -6400.738} C_VEL
LIN {X 0,Y 490.417,Z 826.576,A -85,B 0,C 180,E1 -6401.777,E2 -6401.777} C_VEL
LIN {X 0,Y 490.856,Z 816.131,A -85,B 0,C 180,E1 -6402.633,E2 -6402.633} C_VEL
LIN {X 0,Y 491.119,Z 804.895,A -85,B 0,C 180,E1 -6403.369,E2 -6403.369} C_VEL
LIN {X 0,Y 491.297,Z 793.054,A -85,B 0,C 180,E1 -6403.962,E2 -6403.962} C_VEL
LIN {X 0,Y 491.463,Z 779.72,A -85,B 0,C 180,E1 -6404.433,E2 -6404.433} C_VEL
LIN {X 0,Y 491.488,Z 766.498,A -85,B 0,C 180,E1 -6404.723,E2 -6404.723} C_VEL
LIN {X 0,Y 491.847,Z 700.585,A -85,B 0,C 180,E1 -6405.693,E2 -6405.693} C_VEL
LIN {X 0,Y 488.744,Z 691.605,A -85,B 0,C 180,E1 -6405.948,E2 -6405.948} C_VEL
LIN {X 0,Y 488.726,Z 691.608,A -85,B 0,C 180,E1 -6409.307,E2 -6409.307} C_VEL
LIN {X 0,Y 488.678,Z 691.608,A -85,B 0,C 180,E1 -6411.95,E2 -6411.95} C_VEL
LIN {X 0,Y 488.679,Z 691.614,A -85,B 0,C 180,E1 -6415.035,E2 -6415.035} C_VEL
LIN {X 0,Y 488.704,Z 691.608,A -85,B 0,C 180,E1 -6417.391,E2 -6417.391} C_VEL
LIN {X 0,Y 488.679,Z 691.607,A -85,B 0,C 180,E1 -6420.356,E2 -6420.356} C_VEL
LIN {X 0,Y 488.702,Z 691.611,A -85,B 0,C 180,E1 -6423.478,E2 -6423.478} C_VEL
LIN {X 0,Y 488.65,Z 691.612,A -85,B 0,C 180,E1 -6426.349,E2 -6426.349} C_VEL
LIN {X 0,Y 488.701,Z 691.604,A -85,B 0,C 180,E1 -6429.244,E2 -6429.244} C_VEL
LIN {X 0,Y 488.688,Z 691.608,A -85,B 0,C 180,E1 -6432.515,E2 -6432.515} C_VEL
LIN {X 0,Y 488.663,Z 691.606,A -85,B 0,C 180,E1 -6435.193,E2 -6435.193} C_VEL
LIN {X 0,Y 488.683,Z 691.61,A -85,B 0,C 180,E1 -6437.473,E2 -6437.473} C_VEL
LIN {X 0,Y 488.701,Z 691.604,A -85,B 0,C 180,E1 -6440.745,E2 -6440.745} C_VEL
LIN {X 0,Y 488.627,Z 691.623,A -85,B 0,C 180,E1 -6443.863,E2 -6443.863} C_VEL
LIN {X 0,Y 488.678,Z 691.607,A -85,B 0,C 180,E1 -6446.872,E2 -6446.872} C_VEL
LIN {X 0,Y 488.674,Z 691.612,A -85,B 0,C 180,E1 -6449.777,E2 -6449.777} C_VEL
LIN {X 0,Y 488.732,Z 691.601,A -85,B 0,C 180,E1 -6453.05,E2 -6453.05} C_VEL
LIN {X 0,Y 488.63,Z 691.618,A -85,B 0,C 180,E1 -6456.251,E2 -6456.251} C_VEL
LIN {X 0,Y 488.675,Z 691.609,A -85,B 0,C 180,E1 -6459.172,E2 -6459.172} C_VEL
LIN {X 0,Y 488.663,Z 691.613,A -85,B 0,C 180,E1 -6462.421,E2 -6462.421} C_VEL
LIN {X 0,Y 488.699,Z 691.609,A -85,B 0,C 180,E1 -6464.998,E2 -6464.998} C_VEL
LIN {X 0,Y 488.761,Z 691.602,A -85,B 0,C 180,E1 -6468.386,E2 -6468.386} C_VEL
LIN {X 0,Y 488.749,Z 691.6,A -85,B 0,C 180,E1 -6471.732,E2 -6471.732} C_VEL
LIN {X 0,Y 488.798,Z 691.595,A -85,B 0,C 180,E1 -6474.224,E2 -6474.224} C_VEL
LIN {X 0,Y 488.89,Z 691.583,A -85,B 0,C 180,E1 -6477.528,E2 -6477.528} C_VEL
LIN {X 0,Y 488.888,Z 691.583,A -85,B 0,C 180,E1 -6480,E2 -6480} C_VEL
LIN {X 0,Y 488.891,Z 691.581,A -85,B 0,C 180,E1 -6482.472,E2 -6482.472} C_VEL
LIN {X 0,Y 488.798,Z 691.596,A -85,B 0,C 180,E1 -6485.776,E2 -6485.776} C_VEL
LIN {X 0,Y 488.749,Z 691.598,A -85,B 0,C 180,E1 -6488.268,E2 -6488.268} C_VEL
LIN {X 0,Y 488.761,Z 691.604,A -85,B 0,C 180,E1 -6491.614,E2 -6491.614} C_VEL
LIN {X 0,Y 488.699,Z 691.608,A -85,B 0,C 180,E1 -6495.002,E2 -6495.002} C_VEL
